LIN {X 0,Y 474.319,Z 459.173,A -85,B 0,C 180,E1 -7298.735,E2 -7298.735} C_VEL
LIN {X 0,Y 474.674,Z 450.889,A -85,B 0,C 180,E1 -7300.018,E2 -7300.018} C_VEL
LIN {X 0,Y 475.05,Z 442.392,A -85,B 0,C 180,E1 -7301.088,E2 -7301.088} C_VEL
LIN {X 0,Y 475.606,Z 432.048,A -85,B 0,C 180,E1 -7302.141,E2 -7302.141} C_VEL
LIN {X 0,Y 475.98,Z 420.23,A -85,B 0,C 180,E1 -7303.109,E2 -7303.109} C_VEL
LIN {X 0,Y 476.476,Z 408.181,A -85,B 0,C 180,E1 -7303.867,E2 -7303.867} C_VEL
LIN {X 0,Y 476.914,Z 395.801,A -85,B 0,C 180,E1 -7304.453,E2 -7304.453} C_VEL
LIN {X 0,Y 477.291,Z 383.062,A -85,B 0,C 180,E1 -7304.877,E2 -7304.877} C_VEL
LIN {X 0,Y 477.535,Z 367.874,A -85,B 0,C 180,E1 -7305.17,E2 -7305.17} C_VEL
LIN {X 0,Y 478.066,Z 286.385,A -85,B 0,C 180,E1 -7306.413,E2 -7306.413} C_VEL
LIN {X 0,Y 475.418,Z 270.175,A -85,B 0,C 180,E1 -7306.789,E2 -7306.789} C_VEL
LIN {X 0,Y 475.587,Z 262.703,A -85,B 0,C 180,E1 -7308.078,E2 -7308.078} C_VEL
LIN {X 0,Y 476.357,Z 243.825,A -85,B 0,C 180,E1 -7311.518,E2 -7311.518} C_VEL
LIN {X 0,Y 476.393,Z 237.035,A -85,B 0,C 180,E1 -7312.783,E2 -7312.783} C_VEL
LIN {X 0,Y 474.661,Z 227.951,A -85,B 0,C 180,E1 -7314.637,E2 -7314.637} C_VEL
LIN {X 0,Y 474.679,Z 227.858,A -85,B 0,C 180,E1 -7317.331,E2 -7317.331} C_VEL
LIN {X 0,Y 474.608,Z 227.867,A -85,B 0,C 180,E1 -7320.229,E2 -7320.229} C_VEL
LIN {X 0,Y 474.638,Z 227.86,A -85,B 0,C 180,E1 -7323.219,E2 -7323.219} C_VEL
LIN {X 0,Y 474.587,Z 227.865,A -85,B 0,C 180,E1 -7326.322,E2 -7326.322} C_VEL
LIN {X 0,Y 474.624,Z 227.861,A -85,B 0,C 180,E1 -7329.547,E2 -7329.547} C_VEL
LIN {X 0,Y 474.6,Z 227.87,A -85,B 0,C 180,E1 -7332.231,E2 -7332.231} C_VEL
LIN {X 0,Y 474.618,Z 227.86,A -85,B 0,C 180,E1 -7335.296,E2 -7335.296} C_VEL
LIN {X 0,Y 474.61,Z 227.867,A -85,B 0,C 180,E1 -7338.211,E2 -7338.211} C_VEL
LIN {X 0,Y 474.609,Z 227.858,A -85,B 0,C 180,E1 -7341.54,E2 -7341.54} C_VEL
LIN {X 0,Y 474.619,Z 227.864,A -85,B 0,C 180,E1 -7344.723,E2 -7344.723} C_VEL
LIN {X 0,Y 474.627,Z 227.858,A -85,B 0,C 180,E1 -7347.785,E2 -7347.785} C_VEL
LIN {X 0,Y 474.597,Z 227.868,A -85,B 0,C 180,E1 -7350.888,E2 -7350.888} C_VEL
LIN {X 0,Y 474.588,Z 227.863,A -85,B 0,C 180,E1 -7353.622,E2 -7353.622} C_VEL
LIN {X 0,Y 474.632,Z 227.862,A -85,B 0,C 180,E1 -7356.64,E2 -7356.64} C_VEL
LIN {X 0,Y 474.646,Z 227.856,A -85,B 0,C 180,E1 -7360.087,E2 -7360.087} C_VEL
LIN {X 0,Y 474.628,Z 227.859,A -85,B 0,C 180,E1 -7362.771,E2 -7362.771} C_VEL
LIN {X 0,Y 474.627,Z 227.86,A -85,B 0,C 180,E1 -7365.418,E2 -7365.418} C_VEL
LIN {X 0,Y 474.698,Z 227.849,A -85,B 0,C 180,E1 -7368.035,E2 -7368.035} C_VEL
LIN {X 0,Y 474.66,Z 227.857,A -85,B 0,C 180,E1 -7371.483,E2 -7371.483} C_VEL
LIN {X 0,Y 474.748,Z 227.845,A -85,B 0,C 180,E1 -7374.049,E2 -7374.049} C_VEL
LIN {X 0,Y 474.859,Z 227.833,A -85,B 0,C 180,E1 -7377.452,E2 -7377.452} C_VEL
LIN {X 0,Y 474.865,Z 227.829,A -85,B 0,C 180,E1 -7379.997,E2 -7379.997} C_VEL
LIN {X 0,Y 474.833,Z 227.833,A -85,B 0,C 180,E1 -7382.542,E2 -7382.542} C_VEL
LIN {X 0,Y 474.714,Z 227.852,A -85,B 0,C 180,E1 -7385.945,E2 -7385.945} C_VEL
LIN {X 0,Y 474.65,Z 227.856,A -85,B 0,C 180,E1 -7388.512,E2 -7388.512} C_VEL
LIN {X 0,Y 474.678,Z 227.86,A -85,B 0,C 180,E1 -7391.96,E2 -7391.96} C_VEL
LIN {X 0,Y 474.681,Z 227.855,A -85,B 0,C 180,E1 -7395.453,E2 -7395.453} C_VEL
LIN {X 0,Y 474.642,Z 227.858,A -85,B 0,C 180,E1 -7399.007,E2 -7399.007} C_VEL
LIN {X 0,Y 474.568,Z 227.869,A -85,B 0,C 180,E1 -7401.726,E2 -7401.726} C_VEL
LIN {X 0,Y 474.615,Z 227.865,A -85,B 0,C 180,E1 -7404.491,E2 -7404.491} C_VEL
LIN {X 0,Y 474.614,Z 227.861,A -85,B 0,C 180,E1 -7407.321,E2 -7407.321} C_VEL
LIN {X 0,Y 474.578,Z 227.87,A -85,B 0,C 180,E1 -7410.228,E2 -7410.228} C_VEL
LIN {X 0,Y 474.617,Z 227.862,A -85,B 0,C 180,E1 -7413.217,E2 -7413.217} C_VEL
LIN {X 0,Y 474.566,Z 227.872,A -85,B 0,C 180,E1 -7416.321,E2 -7416.321} C_VEL
LIN {X 0,Y 474.622,Z 227.862,A -85,B 0,C 180,E1 -7419.648,E2 -7419.648} C_VEL
LIN {X 0,Y 474.623,Z 227.867,A -85,B 0,C 180,E1 -7422.928,E2 -7422.928} C_VEL
LIN {X 0,Y 474.644,Z 227.955,A -85,B 0,C 180,E1 -7424.526,E2 -7424.526} C_VEL
LIN {X 0,Y 475.947,Z 235.272,A -85,B 0,C 180,E1 -7426.052,E2 -7426.052} C_VEL
LIN {X 0,Y 475.635,Z 249.047,A -85,B 0,C 180,E1 -7428.661,E2 -7428.661} C_VEL
LIN {X 0,Y 475.424,Z 257.75,A -85,B 0,C 180,E1 -7430.256,E2 -7430.256} C_VEL
LIN {X 0,Y 478.108,Z 273.113,A -85,B 0,C 180,E1 -7430.623,E2 -7430.623} C_VEL
LIN {X 0,Y 477.39,Z 365.589,A -85,B 0,C 180,E1 -7432.055,E2 -7432.055} C_VEL
LIN {X 0,Y 477.099,Z 378.912,A -85,B 0,C 180,E1 -7432.436,E2 -7432.436} C_VEL
LIN {X 0,Y 476.816,Z 391.076,A -85,B 0,C 180,E1 -7432.954,E2 -7432.954} C_VEL
LIN {X 0,Y 476.403,Z 402.075,A -85,B 0,C 180,E1 -7433.576,E2 -7433.576} C_VEL
LIN {X 0,Y 476.121,Z 407.981,A -85,B 0,C 180,E1 -7433.98,E2 -7433.98} C_VEL
LIN {X 0,Y 475.228,Z 413.061,A -85,B 0,C 180,E1 -7434.352,E2 -7434.352} C_VEL
LIN {X 0,Y 472.047,Z 420.996,A -85,B 0,C 180,E1 -7434.971,E2 -7434.971} C_VEL
LIN {X 0,Y 468.888,Z 428.372,A -85,B 0,C 180,E1 -7435.666,E2 -7435.666} C_VEL
LIN {X 0,Y 468.021,Z 432.578,A -85,B 0,C 180,E1 -7436.148,E2 -7436.148} C_VEL
LIN {X 0,Y 467.606,Z 441.038,A -85,B 0,C 180,E1 -7437.308,E2 -7437.308} C_VEL
LIN {X 0,Y 467.237,Z 449.029,A -85,B 0,C 180,E1 -7438.674,E2 -7438.674} C_VEL
LIN {X 0,Y 467.002,Z 455.116,A -85,B 0,C 180,E1 -7439.976,E2 -7439.976} C_VEL
LIN {X 0,Y 466.824,Z 459.697,A -85,B 0,C 180,E1 -7441.201,E2 -7441.201} C_VEL
LIN {X 0,Y 466.694,Z 463.897,A -85,B 0,C 180,E1 -7442.674,E2 -7442.674} C_VEL
LIN {X 0,Y 466.564,Z 466.729,A -85,B 0,C 180,E1 -7444.099,E2 -7444.099} C_VEL
LIN {X 0,Y 466.508,Z 467.992,A -85,B 0,C 180,E1 -7445.051,E2 -7445.051} C_VEL
LIN {X 0,Y 466.486,Z 469.005,A -85,B 0,C 180,E1 -7446.771,E2 -7446.771} C_VEL
LIN {X 0,Y 466.467,Z 468.848,A -85,B 0,C 180,E1 -7447.874,E2 -7447.874} C_VEL
LIN {X 0,Y 466.511,Z 467.954,A -85,B 0,C 180,E1 -7449.059,E2 -7449.059} C_VEL
LIN {X 0,Y 466.617,Z 465.531,A -85,B 0,C 180,E1 -7450.65,E2 -7450.65} C_VEL
LIN {X 0,Y 466.715,Z 462.294,A -85,B 0,C 180,E1 -7452.02,E2 -7452.02} C_VEL
LIN {X 0,Y 466.863,Z 457.92,A -85,B 0,C 180,E1 -7453.381,E2 -7453.381} C_VEL
LIN {X 0,Y 467.122,Z 452.119,A -85,B 0,C 180,E1 -7454.772,E2 -7454.772} C_VEL
LIN {X 0,Y 467.411,Z 445.255,A -85,B 0,C 180,E1 -7456.08,E2 -7456.08} C_VEL
LIN {X 0,Y 467.793,Z 437.03,A -85,B 0,C 180,E1 -7457.34,E2 -7457.34} C_VEL
LIN {X 0,Y 468.253,Z 427.374,A -85,B 0,C 180,E1 -7458.53,E2 -7458.53} C_VEL
LIN {X 0,Y 468.76,Z 417.39,A -85,B 0,C 180,E1 -7459.527,E2 -7459.527} C_VEL
LIN {X 0,Y 469.247,Z 406.384,A -85,B 0,C 180,E1 -7460.409,E2 -7460.409} C_VEL
LIN {X 0,Y 469.753,Z 394.705,A -85,B 0,C 180,E1 -7461.14,E2 -7461.14} C_VEL
LIN {X 0,Y 470.088,Z 382.336,A -85,B 0,C 180,E1 -7461.727,E2 -7461.727} C_VEL
LIN {X 0,Y 470.482,Z 369.805,A -85,B 0,C 180,E1 -7462.14,E2 -7462.14} C_VEL
LIN {X 0,Y 470.668,Z 355.83,A -85,B 0,C 180,E1 -7462.412,E2 -7462.412} C_VEL
LIN {X 0,Y 471.164,Z 272.816,A -85,B 0,C 180,E1 -7463.698,E2 -7463.698} C_VEL
LIN {X 0,Y 468.501,Z 258.149,A -85,B 0,C 180,E1 -7464.054,E2 -7464.054} C_VEL
LIN {X 0,Y 468.635,Z 252.883,A -85,B 0,C 180,E1 -7465.054,E2 -7465.054} C_VEL
LIN {X 0,Y 469.214,Z 238.012,A -85,B 0,C 180,E1 -7468.069,E2 -7468.069} C_VEL
LIN {X 0,Y 467.876,Z 229.061,A -85,B 0,C 180,E1 -7470.001,E2 -7470.001} C_VEL
LIN {X 0,Y 467.826,Z 228.707,A -85,B 0,C 180,E1 -7470.216,E2 -7470.216} C_VEL
LIN {X 0,Y 467.822,Z 228.711,A -85,B 0,C 180,E1 -7472.584,E2 -7472.584} C_VEL
LIN {X 0,Y 467.706,Z 228.723,A -85,B 0,C 180,E1 -7476.039,E2 -7476.039} C_VEL
LIN {X 0,Y 467.644,Z 228.73,A -85,B 0,C 180,E1 -7478.644,E2 -7478.644} C_VEL
LIN {X 0,Y 467.646,Z 228.726,A -85,B 0,C 180,E1 -7482.146,E2 -7482.146} C_VEL
LIN {X 0,Y 467.613,Z 228.737,A -85,B 0,C 180,E1 -7485.887,E2 -7485.887} C_VEL
LIN {X 0,Y 467.588,Z 228.737,A -85,B 0,C 180,E1 -7489.31,E2 -7489.31} C_VEL
LIN {X 0,Y 467.5,Z 228.754,A -85,B 0,C 180,E1 -7492.076,E2 -7492.076} C_VEL
LIN {X 0,Y 467.55,Z 228.739,A -85,B 0,C 180,E1 -7494.891,E2 -7494.891} C_VEL
LIN {X 0,Y 467.548,Z 228.744,A -85,B 0,C 180,E1 -7497.774,E2 -7497.774} C_VEL
LIN {X 0,Y 467.537,Z 228.742,A -85,B 0,C 180,E1 -7501.047,E2 -7501.047} C_VEL
LIN {X 0,Y 467.546,Z 228.744,A -85,B 0,C 180,E1 -7504.243,E2 -7504.243} C_VEL
LIN {X 0,Y 467.493,Z 228.747,A -85,B 0,C 180,E1 -7507.185,E2 -7507.185} C_VEL
LIN {X 0,Y 467.529,Z 228.747,A -85,B 0,C 180,E1 -7510.27,E2 -7510.27} C_VEL
LIN {X 0,Y 467.521,Z 228.738,A -85,B 0,C 180,E1 -7513.749,E2 -7513.749} C_VEL
LIN {X 0,Y 467.521,Z 228.745,A -85,B 0,C 180,E1 -7516.258,E2 -7516.258} C_VEL
LIN {X 0,Y 467.536,Z 228.735,A -85,B 0,C 180,E1 -7519.737,E2 -7519.737} C_VEL
LIN {X 0,Y 467.528,Z 228.739,A -85,B 0,C 180,E1 -7522.818,E2 -7522.818} C_VEL
LIN {X 0,Y 467.56,Z 228.739,A -85,B 0,C 180,E1 -7525.764,E2 -7525.764} C_VEL
LIN {X 0,Y 467.528,Z 228.746,A -85,B 0,C 180,E1 -7528.964,E2 -7528.964} C_VEL
LIN {X 0,Y 467.53,Z 228.731,A -85,B 0,C 180,E1 -7532.23,E2 -7532.23} C_VEL
LIN {X 0,Y 467.542,Z 228.742,A -85,B 0,C 180,E1 -7535.113,E2 -7535.113} C_VEL
LIN {X 0,Y 467.522,Z 228.744,A -85,B 0,C 180,E1 -7537.93,E2 -7537.93} C_VEL
LIN {X 0,Y 467.612,Z 228.724,A -85,B 0,C 180,E1 -7540.696,E2 -7540.696} C_VEL
LIN {X 0,Y 467.632,Z 228.724,A -85,B 0,C 180,E1 -7544.308,E2 -7544.308} C_VEL
LIN {X 0,Y 467.644,Z 228.736,A -85,B 0,C 180,E1 -7547.858,E2 -7547.858} C_VEL
LIN {X 0,Y 467.653,Z 228.725,A -85,B 0,C 180,E1 -7551.36,E2 -7551.36} C_VEL
LIN {X 0,Y 467.701,Z 228.711,A -85,B 0,C 180,E1 -7553.965,E2 -7553.965} C_VEL
LIN {X 0,Y 467.813,Z 228.703,A -85,B 0,C 180,E1 -7557.42,E2 -7557.42} C_VEL
LIN {X 0,Y 467.849,Z 228.708,A -85,B 0,C 180,E1 -7560.003,E2 -7560.003} C_VEL
LIN {X 0,Y 467.814,Z 228.704,A -85,B 0,C 180,E1 -7562.586,E2 -7562.586} C_VEL
LIN {X 0,Y 467.718,Z 228.708,A -85,B 0,C 180,E1 -7566.04,E2 -7566.04} C_VEL
LIN {X 0,Y 467.663,Z 228.732,A -85,B 0,C 180,E1 -7568.646,E2 -7568.646} C_VEL
LIN {X 0,Y 467.662,Z 228.728,A -85,B 0,C 180,E1 -7572.148,E2 -7572.148} C_VEL
LIN {X 0,Y 467.656,Z 228.716,A -85,B 0,C 180,E1 -7575.887,E2 -7575.887} C_VEL
LIN {X 0,Y 467.629,Z 228.733,A -85,B 0,C 180,E1 -7579.31,E2 -7579.31} C_VEL
LIN {X 0,Y 467.539,Z 228.739,A -85,B 0,C 180,E1 -7582.076,E2 -7582.076} C_VEL
LIN {X 0,Y 467.577,Z 228.733,A -85,B 0,C 180,E1 -7584.891,E2 -7584.891} C_VEL
LIN {X 0,Y 467.571,Z 228.738,A -85,B 0,C 180,E1 -7587.774,E2 -7587.774} C_VEL
LIN {X 0,Y 467.574,Z 228.738,A -85,B 0,C 180,E1 -7591.045,E2 -7591.045} C_VEL
LIN {X 0,Y 467.586,Z 228.736,A -85,B 0,C 180,E1 -7594.241,E2 -7594.241} C_VEL
LIN {X 0,Y 467.552,Z 228.743,A -85,B 0,C 180,E1 -7597.186,E2 -7597.186} C_VEL
LIN {X 0,Y 467.569,Z 228.738,A -85,B 0,C 180,E1 -7600.268,E2 -7600.268} C_VEL
LIN {X 0,Y 467.553,Z 228.735,A -85,B 0,C 180,E1 -7602.566,E2 -7602.566} C_VEL
LIN {X 0,Y 467.575,Z 228.739,A -85,B 0,C 180,E1 -7605.053,E2 -7605.053} C_VEL
LIN {X 0,Y 467.574,Z 228.737,A -85,B 0,C 180,E1 -7608.726,E2 -7608.726} C_VEL
LIN {X 0,Y 467.571,Z 228.744,A -85,B 0,C 180,E1 -7611.956,E2 -7611.956} C_VEL
LIN {X 0,Y 467.572,Z 228.739,A -85,B 0,C 180,E1 -7615.168,E2 -7615.168} C_VEL
LIN {X 0,Y 467.592,Z 228.741,A -85,B 0,C 180,E1 -7618.26,E2 -7618.26} C_VEL
LIN {X 0,Y 467.582,Z 228.738,A -85,B 0,C 180,E1 -7621.25,E2 -7621.25} C_VEL
LIN {X 0,Y 467.597,Z 228.743,A -85,B 0,C 180,E1 -7624.159,E2 -7624.159} C_VEL
LIN {X 0,Y 467.654,Z 228.952,A -85,B 0,C 180,E1 -7625.115,E2 -7625.115} C_VEL
LIN {X 0,Y 469.616,Z 239.761,A -85,B 0,C 180,E1 -7627.333,E2 -7627.333} C_VEL
LIN {X 0,Y 469.166,Z 250.64,A -85,B 0,C 180,E1 -7629.388,E2 -7629.388} C_VEL
LIN {X 0,Y 468.53,Z 266.336,A -85,B 0,C 180,E1 -7632.316,E2 -7632.316} C_VEL
LIN {X 0,Y 468.406,Z 270.181,A -85,B 0,C 180,E1 -7632.979,E2 -7632.979} C_VEL
LIN {X 0,Y 471.24,Z 287.662,A -85,B 0,C 180,E1 -7633.384,E2 -7633.384} C_VEL
LIN {X 0,Y 470.546,Z 377.761,A -85,B 0,C 180,E1 -7634.792,E2 -7634.792} C_VEL
LIN {X 0,Y 470.203,Z 391.031,A -85,B 0,C 180,E1 -7635.169,E2 -7635.169} C_VEL
LIN {X 0,Y 469.781,Z 403.762,A -85,B 0,C 180,E1 -7635.709,E2 -7635.709} C_VEL
LIN {X 0,Y 469.301,Z 415.395,A -85,B 0,C 180,E1 -7636.379,E2 -7636.379} C_VEL
LIN {X 0,Y 468.806,Z 426.182,A -85,B 0,C 180,E1 -7637.176,E2 -7637.176} C_VEL
LIN {X 0,Y 468.289,Z 437.241,A -85,B 0,C 180,E1 -7638.2,E2 -7638.2} C_VEL
LIN {X 0,Y 467.866,Z 445.818,A -85,B 0,C 180,E1 -7639.177,E2 -7639.177} C_VEL
LIN {X 0,Y 467.483,Z 453.726,A -85,B 0,C 180,E1 -7640.262,E2 -7640.262} C_VEL
LIN {X 0,Y 467.154,Z 461.449,A -85,B 0,C 180,E1 -7641.565,E2 -7641.565} C_VEL
LIN {X 0,Y 466.86,Z 468.553,A -85,B 0,C 180,E1 -7643.082,E2 -7643.082} C_VEL
LIN {X 0,Y 466.792,Z 473.281,A -85,B 0,C 180,E1 -7644.383,E2 -7644.383} C_VEL
LIN {X 0,Y 466.649,Z 476.891,A -85,B 0,C 180,E1 -7645.681,E2 -7645.681} C_VEL
LIN {X 0,Y 466.663,Z 478.755,A -85,B 0,C 180,E1 -7646.546,E2 -7646.546} C_VEL
LIN {X 0,Y 466.646,Z 480.152,A -85,B 0,C 180,E1 -7647.41,E2 -7647.41} C_VEL
LIN {X 0,Y 466.591,Z 481.755,A -85,B 0,C 180,E1 -7649.136,E2 -7649.136} C_VEL
LIN {X 0,Y 466.601,Z 481.973,A -85,B 0,C 180,E1 -7649.999,E2 -7649.999} C_VEL
LIN {X 0,Y 466.606,Z 481.151,A -85,B 0,C 180,E1 -7651.726,E2 -7651.726} C_VEL
LIN {X 0,Y 466.646,Z 480.157,A -85,B 0,C 180,E1 -7652.589,E2 -7652.589} C_VEL
LIN {X 0,Y 466.663,Z 478.763,A -85,B 0,C 180,E1 -7653.453,E2 -7653.453} C_VEL
LIN {X 0,Y 466.693,Z 475.829,A -85,B 0,C 180,E1 -7654.75,E2 -7654.75} C_VEL
LIN {X 0,Y 466.78,Z 471.859,A -85,B 0,C 180,E1 -7656.049,E2 -7656.049} C_VEL
LIN {X 0,Y 466.981,Z 465.754,A -85,B 0,C 180,E1 -7657.566,E2 -7657.566} C_VEL
LIN {X 0,Y 467.282,Z 459.082,A -85,B 0,C 180,E1 -7658.867,E2 -7658.867} C_VEL
LIN {X 0,Y 467.63,Z 450.802,A -85,B 0,C 180,E1 -7660.17,E2 -7660.17} C_VEL
LIN {X 0,Y 468.068,Z 442.312,A -85,B 0,C 180,E1 -7661.255,E2 -7661.255} C_VEL
LIN {X 0,Y 468.648,Z 432.148,A -85,B 0,C 180,E1 -7662.308,E2 -7662.308} C_VEL
LIN {X 0,Y 468.971,Z 421.726,A -85,B 0,C 180,E1 -7663.188,E2 -7663.188} C_VEL
LIN {X 0,Y 469.522,Z 410.055,A -85,B 0,C 180,E1 -7663.966,E2 -7663.966} C_VEL
LIN {X 0,Y 469.958,Z 398.351,A -85,B 0,C 180,E1 -7664.561,E2 -7664.561} C_VEL
LIN {X 0,Y 470.425,Z 384.874,A -85,B 0,C 180,E1 -7665.044,E2 -7665.044} C_VEL
LIN {X 0,Y 470.647,Z 371.473,A -85,B 0,C 180,E1 -7665.342,E2 -7665.342} C_VEL
LIN {X 0,Y 471.274,Z 287.31,A -85,B 0,C 180,E1 -7666.643,E2 -7666.643} C_VEL
LIN {X 0,Y 468.443,Z 270.181,A -85,B 0,C 180,E1 -7667.044,E2 -7667.044} C_VEL
LIN {X 0,Y 468.441,Z 267.494,A -85,B 0,C 180,E1 -7667.46,E2 -7667.46} C_VEL
LIN {X 0,Y 469.125,Z 250.395,A -85,B 0,C 180,E1 -7670.612,E2 -7670.612} C_VEL
LIN {X 0,Y 469.575,Z 239.398,A -85,B 0,C 180,E1 -7672.667,E2 -7672.667} C_VEL
LIN {X 0,Y 467.644,Z 228.871,A -85,B 0,C 180,E1 -7674.825,E2 -7674.825} C_VEL
LIN {X 0,Y 467.621,Z 228.739,A -85,B 0,C 180,E1 -7677.768,E2 -7677.768} C_VEL
LIN {X 0,Y 467.571,Z 228.741,A -85,B 0,C 180,E1 -7681.043,E2 -7681.043} C_VEL
LIN {X 0,Y 467.592,Z 228.741,A -85,B 0,C 180,E1 -7684.24,E2 -7684.24} C_VEL
LIN {X 0,Y 467.545,Z 228.739,A -85,B 0,C 180,E1 -7687.184,E2 -7687.184} C_VEL
LIN {X 0,Y 467.562,Z 228.74,A -85,B 0,C 180,E1 -7690.265,E2 -7690.265} C_VEL
LIN {X 0,Y 467.563,Z 228.742,A -85,B 0,C 180,E1 -7692.562,E2 -7692.562} C_VEL
LIN {X 0,Y 467.567,Z 228.739,A -85,B 0,C 180,E1 -7695.051,E2 -7695.051} C_VEL
LIN {X 0,Y 467.568,Z 228.744,A -85,B 0,C 180,E1 -7698.594,E2 -7698.594} C_VEL
LIN {X 0,Y 467.562,Z 228.738,A -85,B 0,C 180,E1 -7701.953,E2 -7701.953} C_VEL
LIN {X 0,Y 467.556,Z 228.74,A -85,B 0,C 180,E1 -7705.164,E2 -7705.164} C_VEL
LIN {X 0,Y 467.577,Z 228.74,A -85,B 0,C 180,E1 -7708.257,E2 -7708.257} C_VEL
LIN {X 0,Y 467.543,Z 228.742,A -85,B 0,C 180,E1 -7711.246,E2 -7711.246} C_VEL
LIN {X 0,Y 467.576,Z 228.739,A -85,B 0,C 180,E1 -7714.399,E2 -7714.399} C_VEL
LIN {X 0,Y 467.57,Z 228.74,A -85,B 0,C 180,E1 -7716.993,E2 -7716.993} C_VEL
LIN {X 0,Y 467.617,Z 228.732,A -85,B 0,C 180,E1 -7719.775,E2 -7719.775} C_VEL
LIN {X 0,Y 467.589,Z 228.733,A -85,B 0,C 180,E1 -7722.504,E2 -7722.504} C_VEL
LIN {X 0,Y 467.589,Z 228.74,A -85,B 0,C 180,E1 -7725.193,E2 -7725.193} C_VEL
LIN {X 0,Y 467.65,Z 228.728,A -85,B 0,C 180,E1 -7727.852,E2 -7727.852} C_VEL
LIN {X 0,Y 467.629,Z 228.732,A -85,B 0,C 180,E1 -7731.354,E2 -7731.354} C_VEL
LIN {X 0,Y 467.713,Z 228.722,A -85,B 0,C 180,E1 -7733.959,E2 -7733.959} C_VEL
LIN {X 0,Y 467.8,Z 228.712,A -85,B 0,C 180,E1 -7737.414,E2 -7737.414} C_VEL
LIN {X 0,Y 467.814,Z 228.707,A -85,B 0,C 180,E1 -7739.997,E2 -7739.997} C_VEL
LIN {X 0,Y 467.777,Z 228.712,A -85,B 0,C 180,E1 -7742.58,E2 -7742.58} C_VEL
LIN {X 0,Y 467.679,Z 228.728,A -85,B 0,C 180,E1 -7746.035,E2 -7746.035} C_VEL
LIN {X 0,Y 467.619,Z 228.731,A -85,B 0,C 180,E1 -7748.641,E2 -7748.641} C_VEL
LIN {X 0,Y 467.632,Z 228.735,A -85,B 0,C 180,E1 -7752.143,E2 -7752.143} C_VEL
LIN {X 0,Y 467.621,Z 228.737,A -85,B 0,C 180,E1 -7755.692,E2 -7755.692} C_VEL
LIN {X 0,Y 467.601,Z 228.735,A -85,B 0,C 180,E1 -7759.305,E2 -7759.305} C_VEL
LIN {X 0,Y 467.515,Z 228.753,A -85,B 0,C 180,E1 -7762.071,E2 -7762.071} C_VEL
LIN {X 0,Y 467.562,Z 228.739,A -85,B 0,C 180,E1 -7764.886,E2 -7764.886} C_VEL
LIN {X 0,Y 467.558,Z 228.742,A -85,B 0,C 180,E1 -7767.769,E2 -7767.769} C_VEL
LIN {X 0,Y 467.543,Z 228.743,A -85,B 0,C 180,E1 -7771.042,E2 -7771.042} C_VEL
LIN {X 0,Y 467.564,Z 228.745,A -85,B 0,C 180,E1 -7774.24,E2 -7774.24} C_VEL
LIN {X 0,Y 467.523,Z 228.746,A -85,B 0,C 180,E1 -7777.184,E2 -7777.184} C_VEL
LIN {X 0,Y 467.568,Z 228.744,A -85,B 0,C 180,E1 -7780.26,E2 -7780.26} C_VEL
LIN {X 0,Y 467.59,Z 228.742,A -85,B 0,C 180,E1 -7782.569,E2 -7782.569} C_VEL
LIN {X 0,Y 467.591,Z 228.848,A -85,B 0,C 180,E1 -7784.341,E2 -7784.341} C_VEL
LIN {X 0,Y 469.033,Z 236.661,A -85,B 0,C 180,E1 -7785.985,E2 -7785.985} C_VEL
LIN {X 0,Y 468.672,Z 250.101,A -85,B 0,C 180,E1 -7788.564,E2 -7788.564} C_VEL
LIN {X 0,Y 468.47,Z 257.854,A -85,B 0,C 180,E1 -7789.993,E2 -7789.993} C_VEL
LIN {X 0,Y 470.658,Z 269.971,A -85,B 0,C 180,E1 -7790.3,E2 -7790.3} C_VEL
LIN {X 0,Y 471.343,Z 275.192,A -85,B 0,C 180,E1 -7790.409,E2 -7790.409} C_VEL
LIN {X 0,Y 470.548,Z 365.863,A -85,B 0,C 180,E1 -7791.833,E2 -7791.833} C_VEL
LIN {X 0,Y 470.245,Z 379.37,A -85,B 0,C 180,E1 -7792.23,E2 -7792.23} C_VEL
LIN {X 0,Y 469.899,Z 392.099,A -85,B 0,C 180,E1 -7792.787,E2 -7792.787} C_VEL
LIN {X 0,Y 469.448,Z 403.23,A -85,B 0,C 180,E1 -7793.443,E2 -7793.443} C_VEL
LIN {X 0,Y 468.858,Z 415.313,A -85,B 0,C 180,E1 -7794.359,E2 -7794.359} C_VEL
LIN {X 0,Y 468.382,Z 425.748,A -85,B 0,C 180,E1 -7795.358,E2 -7795.358} C_VEL
LIN {X 0,Y 468.021,Z 432.578,A -85,B 0,C 180,E1 -7796.148,E2 -7796.148} C_VEL
LIN {X 0,Y 467.149,Z 436.69,A -85,B 0,C 180,E1 -7796.659,E2 -7796.659} C_VEL
LIN {X 0,Y 463.971,Z 443.007,A -85,B 0,C 180,E1 -7797.519,E2 -7797.519} C_VEL
LIN {X 0,Y 460.852,Z 448.667,A -85,B 0,C 180,E1 -7798.452,E2 -7798.452} C_VEL
LIN {X 0,Y 460.083,Z 451.747,A -85,B 0,C 180,E1 -7799.073,E2 -7799.073} C_VEL
LIN {X 0,Y 459.818,Z 458.017,A -85,B 0,C 180,E1 -7800.589,E2 -7800.589} C_VEL
LIN {X 0,Y 459.649,Z 462.837,A -85,B 0,C 180,E1 -7802.13,E2 -7802.13} C_VEL
LIN {X 0,Y 459.496,Z 466.202,A -85,B 0,C 180,E1 -7803.67,E2 -7803.67} C_VEL
LIN {X 0,Y 459.448,Z 467.646,A -85,B 0,C 180,E1 -7804.641,E2 -7804.641} C_VEL
LIN {X 0,Y 459.388,Z 468.621,A -85,B 0,C 180,E1 -7805.604,E2 -7805.604} C_VEL
LIN {X 0,Y 459.385,Z 469.077,A -85,B 0,C 180,E1 -7806.612,E2 -7806.612} C_VEL
LIN {X 0,Y 459.369,Z 469.065,A -85,B 0,C 180,E1 -7807.514,E2 -7807.514} C_VEL
LIN {X 0,Y 459.42,Z 468.206,A -85,B 0,C 180,E1 -7808.918,E2 -7808.918} C_VEL
LIN {X 0,Y 459.508,Z 466.289,A -85,B 0,C 180,E1 -7810.338,E2 -7810.338} C_VEL
LIN {X 0,Y 459.601,Z 464.045,A -85,B 0,C 180,E1 -7811.44,E2 -7811.44} C_VEL
LIN {X 0,Y 459.738,Z 459.279,A -85,B 0,C 180,E1 -7813.116,E2 -7813.116} C_VEL
LIN {X 0,Y 460.015,Z 453.486,A -85,B 0,C 180,E1 -7814.609,E2 -7814.609} C_VEL
LIN {X 0,Y 460.337,Z 446.061,A -85,B 0,C 180,E1 -7816.087,E2 -7816.087} C_VEL
LIN {X 0,Y 460.768,Z 437.468,A -85,B 0,C 180,E1 -7817.446,E2 -7817.446} C_VEL
LIN {X 0,Y 461.216,Z 428.58,A -85,B 0,C 180,E1 -7818.575,E2 -7818.575} C_VEL
LIN {X 0,Y 461.806,Z 417.615,A -85,B 0,C 180,E1 -7819.7,E2 -7819.7} C_VEL
LIN {X 0,Y 462.317,Z 407.003,A -85,B 0,C 180,E1 -7820.57,E2 -7820.57} C_VEL
LIN {X 0,Y 462.842,Z 395.275,A -85,B 0,C 180,E1 -7821.322,E2 -7821.322} C_VEL
LIN {X 0,Y 463.211,Z 382.698,A -85,B 0,C 180,E1 -7821.933,E2 -7821.933} C_VEL
LIN {X 0,Y 463.64,Z 370.292,A -85,B 0,C 180,E1 -7822.352,E2 -7822.352} C_VEL
LIN {X 0,Y 463.817,Z 356.646,A -85,B 0,C 180,E1 -7822.628,E2 -7822.628} C_VEL
LIN {X 0,Y 464.339,Z 273.699,A -85,B 0,C 180,E1 -7823.933,E2 -7823.933} C_VEL
LIN {X 0,Y 461.578,Z 258.553,A -85,B 0,C 180,E1 -7824.294,E2 -7824.294} C_VEL
LIN {X 0,Y 461.552,Z 257.413,A -85,B 0,C 180,E1 -7824.43,E2 -7824.43} C_VEL
LIN {X 0,Y 462.272,Z 240.826,A -85,B 0,C 180,E1 -7827.823,E2 -7827.823} C_VEL
LIN {X 0,Y 461.62,Z 234.738,A -85,B 0,C 180,E1 -7829.128,E2 -7829.128} C_VEL
LIN {X 0,Y 460.796,Z 229.649,A -85,B 0,C 180,E1 -7830.301,E2 -7830.301} C_VEL
LIN {X 0,Y 460.788,Z 229.588,A -85,B 0,C 180,E1 -7832.623,E2 -7832.623} C_VEL
LIN {X 0,Y 460.671,Z 229.599,A -85,B 0,C 180,E1 -7836.131,E2 -7836.131} C_VEL
LIN {X 0,Y 460.591,Z 229.609,A -85,B 0,C 180,E1 -7838.778,E2 -7838.778} C_VEL
LIN {X 0,Y 460.598,Z 229.602,A -85,B 0,C 180,E1 -7842.458,E2 -7842.458} C_VEL
LIN {X 0,Y 460.565,Z 229.614,A -85,B 0,C 180,E1 -7845.999,E2 -7845.999} C_VEL
LIN {X 0,Y 460.536,Z 229.614,A -85,B 0,C 180,E1 -7848.903,E2 -7848.903} C_VEL
LIN {X 0,Y 460.482,Z 229.622,A -85,B 0,C 180,E1 -7851.488,E2 -7851.488} C_VEL
LIN {X 0,Y 460.496,Z 229.622,A -85,B 0,C 180,E1 -7854.335,E2 -7854.335} C_VEL
LIN {X 0,Y 460.502,Z 229.618,A -85,B 0,C 180,E1 -7857.249,E2 -7857.249} C_VEL
LIN {X 0,Y 460.476,Z 229.623,A -85,B 0,C 180,E1 -7860.243,E2 -7860.243} C_VEL
LIN {X 0,Y 460.487,Z 229.619,A -85,B 0,C 180,E1 -7863.329,E2 -7863.329} C_VEL
LIN {X 0,Y 460.436,Z 229.629,A -85,B 0,C 180,E1 -7866.534,E2 -7866.534} C_VEL
LIN {X 0,Y 460.483,Z 229.621,A -85,B 0,C 180,E1 -7869.868,E2 -7869.868} C_VEL
LIN {X 0,Y 460.442,Z 229.623,A -85,B 0,C 180,E1 -7872.897,E2 -7872.897} C_VEL
LIN {X 0,Y 460.48,Z 229.62,A -85,B 0,C 180,E1 -7875.835,E2 -7875.835} C_VEL
LIN {X 0,Y 460.493,Z 229.619,A -85,B 0,C 180,E1 -7878.99,E2 -7878.99} C_VEL
LIN {X 0,Y 460.481,Z 229.611,A -85,B 0,C 180,E1 -7882.38,E2 -7882.38} C_VEL
LIN {X 0,Y 460.519,Z 229.617,A -85,B 0,C 180,E1 -7885.626,E2 -7885.626} C_VEL
LIN {X 0,Y 460.489,Z 229.62,A -85,B 0,C 180,E1 -7888.746,E2 -7888.746} C_VEL
LIN {X 0,Y 460.491,Z 229.61,A -85,B 0,C 180,E1 -7891.767,E2 -7891.767} C_VEL
LIN {X 0,Y 460.5,Z 229.616,A -85,B 0,C 180,E1 -7894.706,E2 -7894.706} C_VEL
LIN {X 0,Y 460.498,Z 229.624,A -85,B 0,C 180,E1 -7897.575,E2 -7897.575} C_VEL
LIN {X 0,Y 460.559,Z 229.603,A -85,B 0,C 180,E1 -7900.388,E2 -7900.388} C_VEL
LIN {X 0,Y 460.599,Z 229.602,A -85,B 0,C 180,E1 -7904.062,E2 -7904.062} C_VEL
LIN {X 0,Y 460.599,Z 229.611,A -85,B 0,C 180,E1 -7907.669,E2 -7907.669} C_VEL
LIN {X 0,Y 460.602,Z 229.602,A -85,B 0,C 180,E1 -7911.227,E2 -7911.227} C_VEL
LIN {X 0,Y 460.667,Z 229.587,A -85,B 0,C 180,E1 -7913.873,E2 -7913.873} C_VEL
LIN {X 0,Y 460.757,Z 229.582,A -85,B 0,C 180,E1 -7917.38,E2 -7917.38} C_VEL
LIN {X 0,Y 460.819,Z 229.584,A -85,B 0,C 180,E1 -7920.003,E2 -7920.003} C_VEL
LIN {X 0,Y 460.758,Z 229.582,A -85,B 0,C 180,E1 -7922.626,E2 -7922.626} C_VEL
LIN {X 0,Y 460.685,Z 229.584,A -85,B 0,C 180,E1 -7926.133,E2 -7926.133} C_VEL
LIN {X 0,Y 460.612,Z 229.608,A -85,B 0,C 180,E1 -7928.779,E2 -7928.779} C_VEL
LIN {X 0,Y 460.603,Z 229.611,A -85,B 0,C 180,E1 -7932.437,E2 -7932.437} C_VEL
LIN {X 0,Y 460.609,Z 229.594,A -85,B 0,C 180,E1 -7936,E2 -7936} C_VEL
LIN {X 0,Y 460.575,Z 229.609,A -85,B 0,C 180,E1 -7939.618,E2 -7939.618} C_VEL
LIN {X 0,Y 460.516,Z 229.616,A -85,B 0,C 180,E1 -7942.431,E2 -7942.431} C_VEL
LIN {X 0,Y 460.556,Z 229.609,A -85,B 0,C 180,E1 -7945.798,E2 -7945.798} C_VEL
LIN {X 0,Y 460.524,Z 229.616,A -85,B 0,C 180,E1 -7948.237,E2 -7948.237} C_VEL
LIN {X 0,Y 460.53,Z 229.614,A -85,B 0,C 180,E1 -7951.284,E2 -7951.284} C_VEL
LIN {X 0,Y 460.531,Z 229.615,A -85,B 0,C 180,E1 -7954.505,E2 -7954.505} C_VEL
LIN {X 0,Y 460.508,Z 229.619,A -85,B 0,C 180,E1 -7957.625,E2 -7957.625} C_VEL
LIN {X 0,Y 460.529,Z 229.617,A -85,B 0,C 180,E1 -7961.014,E2 -7961.014} C_VEL
LIN {X 0,Y 460.521,Z 229.616,A -85,B 0,C 180,E1 -7964.59,E2 -7964.59} C_VEL
LIN {X 0,Y 460.501,Z 229.626,A -85,B 0,C 180,E1 -7967.816,E2 -7967.816} C_VEL
LIN {X 0,Y 460.523,Z 229.621,A -85,B 0,C 180,E1 -7970.136,E2 -7970.136} C_VEL
LIN {X 0,Y 460.482,Z 229.625,A -85,B 0,C 180,E1 -7973.471,E2 -7973.471} C_VEL
LIN {X 0,Y 460.538,Z 229.614,A -85,B 0,C 180,E1 -7976.675,E2 -7976.675} C_VEL
LIN {X 0,Y 460.519,Z 229.619,A -85,B 0,C 180,E1 -7979.76,E2 -7979.76} C_VEL
LIN {X 0,Y 460.568,Z 229.614,A -85,B 0,C 180,E1 -7982.755,E2 -7982.755} C_VEL
LIN {X 0,Y 460.557,Z 229.65,A -85,B 0,C 180,E1 -7984.826,E2 -7984.826} C_VEL
LIN {X 0,Y 461.108,Z 232.34,A -85,B 0,C 180,E1 -7985.459,E2 -7985.459} C_VEL
LIN {X 0,Y 462.73,Z 242.061,A -85,B 0,C 180,E1 -7987.449,E2 -7987.449} C_VEL
LIN {X 0,Y 461.825,Z 260.689,A -85,B 0,C 180,E1 -7990.997,E2 -7990.997} C_VEL
LIN {X 0,Y 461.435,Z 269.989,A -85,B 0,C 180,E1 -7992.714,E2 -7992.714} C_VEL
LIN {X 0,Y 463.43,Z 282.062,A -85,B 0,C 180,E1 -7993.013,E2 -7993.013} C_VEL
LIN {X 0,Y 464.429,Z 289.288,A -85,B 0,C 180,E1 -7993.165,E2 -7993.165} C_VEL
LIN {X 0,Y 463.695,Z 377.425,A -85,B 0,C 180,E1 -7994.562,E2 -7994.562} C_VEL
LIN {X 0,Y 463.318,Z 390.777,A -85,B 0,C 180,E1 -7994.943,E2 -7994.943} C_VEL
LIN {X 0,Y 462.88,Z 403.548,A -85,B 0,C 180,E1 -7995.491,E2 -7995.491} C_VEL
LIN {X 0,Y 462.396,Z 414.894,A -85,B 0,C 180,E1 -7996.149,E2 -7996.149} C_VEL
LIN {X 0,Y 461.81,Z 426.973,A -85,B 0,C 180,E1 -7997.061,E2 -7997.061} C_VEL
LIN {X 0,Y 461.26,Z 438.152,A -85,B 0,C 180,E1 -7998.129,E2 -7998.129} C_VEL
LIN {X 0,Y 460.784,Z 447.374,A -85,B 0,C 180,E1 -7999.231,E2 -7999.231} C_VEL
LIN {X 0,Y 460.326,Z 456.343,A -85,B 0,C 180,E1 -8000.553,E2 -8000.553} C_VEL
LIN {X 0,Y 460.016,Z 463.564,A -85,B 0,C 180,E1 -8001.875,E2 -8001.875} C_VEL
LIN {X 0,Y 459.782,Z 468.434,A -85,B 0,C 180,E1 -8002.975,E2 -8002.975} C_VEL
LIN {X 0,Y 459.711,Z 473.168,A -85,B 0,C 180,E1 -8004.296,E2 -8004.296} C_VEL
LIN {X 0,Y 459.567,Z 476.783,A -85,B 0,C 180,E1 -8005.614,E2 -8005.614} C_VEL
LIN {X 0,Y 459.56,Z 478.649,A -85,B 0,C 180,E1 -8006.492,E2 -8006.492} C_VEL
LIN {X 0,Y 459.569,Z 480.05,A -85,B 0,C 180,E1 -8007.37,E2 -8007.37} C_VEL
LIN {X 0,Y 459.497,Z 481.655,A -85,B 0,C 180,E1 -8009.123,E2 -8009.123} C_VEL
LIN {X 0,Y 459.503,Z 481.875,A -85,B 0,C 180,E1 -8009.999,E2 -8009.999} C_VEL
LIN {X 0,Y 459.518,Z 481.055,A -85,B 0,C 180,E1 -8011.752,E2 -8011.752} C_VEL
LIN {X 0,Y 459.569,Z 480.062,A -85,B 0,C 180,E1 -8012.629,E2 -8012.629} C_VEL
LIN {X 0,Y 459.559,Z 478.669,A -85,B 0,C 180,E1 -8013.506,E2 -8013.506} C_VEL
LIN {X 0,Y 459.625,Z 475.738,A -85,B 0,C 180,E1 -8014.823,E2 -8014.823} C_VEL
LIN {X 0,Y 459.719,Z 470.744,A -85,B 0,C 180,E1 -8016.429,E2 -8016.429} C_VEL
LIN {X 0,Y 459.961,Z 464.655,A -85,B 0,C 180,E1 -8017.903,E2 -8017.903} C_VEL
LIN {X 0,Y 460.257,Z 457.759,A -85,B 0,C 180,E1 -8019.225,E2 -8019.225} C_VEL
LIN {X 0,Y 460.664,Z 449.13,A -85,B 0,C 180,E1 -8020.548,E2 -8020.548} C_VEL
LIN {X 0,Y 461.229,Z 440.281,A -85,B 0,C 180,E1 -8021.647,E2 -8021.647} C_VEL
LIN {X 0,Y 461.765,Z 430.434,A -85,B 0,C 180,E1 -8022.65,E2 -8022.65} C_VEL
LIN {X 0,Y 462.159,Z 419.937,A -85,B 0,C 180,E1 -8023.52,E2 -8023.52} C_VEL
LIN {X 0,Y 462.714,Z 408.058,A -85,B 0,C 180,E1 -8024.288,E2 -8024.288} C_VEL
LIN {X 0,Y 463.177,Z 395.703,A -85,B 0,C 180,E1 -8024.891,E2 -8024.891} C_VEL
LIN {X 0,Y 463.619,Z 383.02,A -85,B 0,C 180,E1 -8025.327,E2 -8025.327} C_VEL
LIN {X 0,Y 463.887,Z 367.977,A -85,B 0,C 180,E1 -8025.627,E2 -8025.627} C_VEL
LIN {X 0,Y 464.383,Z 287.569,A -85,B 0,C 180,E1 -8026.895,E2 -8026.895} C_VEL
LIN {X 0,Y 461.5,Z 270.264,A -85,B 0,C 180,E1 -8027.302,E2 -8027.302} C_VEL
LIN {X 0,Y 461.459,Z 268.512,A -85,B 0,C 180,E1 -8027.527,E2 -8027.527} C_VEL
LIN {X 0,Y 462.153,Z 251.534,A -85,B 0,C 180,E1 -8030.705,E2 -8030.705} C_VEL
LIN {X 0,Y 462.666,Z 241.763,A -85,B 0,C 180,E1 -8032.553,E2 -8032.553} C_VEL
LIN {X 0,Y 461.918,Z 236.377,A -85,B 0,C 180,E1 -8033.635,E2 -8033.635} C_VEL
LIN {X 0,Y 460.565,Z 229.731,A -85,B 0,C 180,E1 -8035.052,E2 -8035.052} C_VEL
LIN {X 0,Y 460.554,Z 229.617,A -85,B 0,C 180,E1 -8038.232,E2 -8038.232} C_VEL
LIN {X 0,Y 460.525,Z 229.62,A -85,B 0,C 180,E1 -8041.281,E2 -8041.281} C_VEL
LIN {X 0,Y 460.535,Z 229.618,A -85,B 0,C 180,E1 -8044.504,E2 -8044.504} C_VEL
LIN {X 0,Y 460.501,Z 229.619,A -85,B 0,C 180,E1 -8047.622,E2 -8047.622} C_VEL
LIN {X 0,Y 460.522,Z 229.615,A -85,B 0,C 180,E1 -8051.011,E2 -8051.011} C_VEL
LIN {X 0,Y 460.507,Z 229.624,A -85,B 0,C 180,E1 -8054.167,E2 -8054.167} C_VEL
LIN {X 0,Y 460.494,Z 229.621,A -85,B 0,C 180,E1 -8057.101,E2 -8057.101} C_VEL
LIN {X 0,Y 460.515,Z 229.622,A -85,B 0,C 180,E1 -8060.134,E2 -8060.134} C_VEL
LIN {X 0,Y 460.473,Z 229.622,A -85,B 0,C 180,E1 -8063.468,E2 -8063.468} C_VEL
LIN {X 0,Y 460.516,Z 229.624,A -85,B 0,C 180,E1 -8066.672,E2 -8066.672} C_VEL
LIN {X 0,Y 460.503,Z 229.618,A -85,B 0,C 180,E1 -8069.757,E2 -8069.757} C_VEL
LIN {X 0,Y 460.49,Z 229.623,A -85,B 0,C 180,E1 -8072.749,E2 -8072.749} C_VEL
LIN {X 0,Y 460.516,Z 229.616,A -85,B 0,C 180,E1 -8075.664,E2 -8075.664} C_VEL
LIN {X 0,Y 460.519,Z 229.618,A -85,B 0,C 180,E1 -8078.576,E2 -8078.576} C_VEL
LIN {X 0,Y 460.58,Z 229.608,A -85,B 0,C 180,E1 -8081.308,E2 -8081.308} C_VEL
LIN {X 0,Y 460.601,Z 229.606,A -85,B 0,C 180,E1 -8084.056,E2 -8084.056} C_VEL
LIN {X 0,Y 460.604,Z 229.608,A -85,B 0,C 180,E1 -8087.663,E2 -8087.663} C_VEL
LIN {X 0,Y 460.584,Z 229.61,A -85,B 0,C 180,E1 -8091.22,E2 -8091.22} C_VEL
LIN {X 0,Y 460.679,Z 229.599,A -85,B 0,C 180,E1 -8093.867,E2 -8093.867} C_VEL
LIN {X 0,Y 460.744,Z 229.59,A -85,B 0,C 180,E1 -8097.374,E2 -8097.374} C_VEL
LIN {X 0,Y 460.764,Z 229.585,A -85,B 0,C 180,E1 -8099.997,E2 -8099.997} C_VEL
LIN {X 0,Y 460.725,Z 229.59,A -85,B 0,C 180,E1 -8102.62,E2 -8102.62} C_VEL
LIN {X 0,Y 460.646,Z 229.603,A -85,B 0,C 180,E1 -8106.128,E2 -8106.128} C_VEL
LIN {X 0,Y 460.574,Z 229.609,A -85,B 0,C 180,E1 -8108.774,E2 -8108.774} C_VEL
LIN {X 0,Y 460.582,Z 229.61,A -85,B 0,C 180,E1 -8112.432,E2 -8112.432} C_VEL
LIN {X 0,Y 460.584,Z 229.615,A -85,B 0,C 180,E1 -8115.994,E2 -8115.994} C_VEL
LIN {X 0,Y 460.548,Z 229.616,A -85,B 0,C 180,E1 -8119.613,E2 -8119.613} C_VEL
LIN {X 0,Y 460.491,Z 229.624,A -85,B 0,C 180,E1 -8122.426,E2 -8122.426} C_VEL
LIN {X 0,Y 460.527,Z 229.617,A -85,B 0,C 180,E1 -8125.794,E2 -8125.794} C_VEL
LIN {X 0,Y 460.504,Z 229.62,A -85,B 0,C 180,E1 -8128.232,E2 -8128.232} C_VEL
LIN {X 0,Y 460.495,Z 229.62,A -85,B 0,C 180,E1 -8131.28,E2 -8131.28} C_VEL
LIN {X 0,Y 460.508,Z 229.623,A -85,B 0,C 180,E1 -8134.503,E2 -8134.503} C_VEL
LIN {X 0,Y 460.502,Z 229.619,A -85,B 0,C 180,E1 -8137.618,E2 -8137.618} C_VEL
LIN {X 0,Y 460.53,Z 229.621,A -85,B 0,C 180,E1 -8140.269,E2 -8140.269} C_VEL
LIN {X 0,Y 460.504,Z 229.625,A -85,B 0,C 180,E1 -8143.369,E2 -8143.369} C_VEL
LIN {X 0,Y 460.559,Z 229.805,A -85,B 0,C 180,E1 -8144.177,E2 -8144.177} C_VEL
LIN {X 0,Y 462.09,Z 238.053,A -85,B 0,C 180,E1 -8145.918,E2 -8145.918} C_VEL
LIN {X 0,Y 461.693,Z 251.531,A -85,B 0,C 180,E1 -8148.536,E2 -8148.536} C_VEL
LIN {X 0,Y 461.51,Z 257.896,A -85,B 0,C 180,E1 -8149.716,E2 -8149.716} C_VEL
LIN {X 0,Y 462.456,Z 263.011,A -85,B 0,C 180,E1 -8149.875,E2 -8149.875} C_VEL
LIN {X 0,Y 464.563,Z 276.017,A -85,B 0,C 180,E1 -8150.167,E2 -8150.167} C_VEL
LIN {X 0,Y 463.712,Z 366.016,A -85,B 0,C 180,E1 -8151.603,E2 -8151.603} C_VEL
LIN {X 0,Y 463.393,Z 379.034,A -85,B 0,C 180,E1 -8151.987,E2 -8151.987} C_VEL
LIN {X 0,Y 463.069,Z 391.264,A -85,B 0,C 180,E1 -8152.521,E2 -8152.521} C_VEL
LIN {X 0,Y 462.54,Z 403.626,A -85,B 0,C 180,E1 -8153.255,E2 -8153.255} C_VEL
LIN {X 0,Y 461.935,Z 415.206,A -85,B 0,C 180,E1 -8154.145,E2 -8154.145} C_VEL
LIN {X 0,Y 461.46,Z 424.543,A -85,B 0,C 180,E1 -8155.039,E2 -8155.039} C_VEL
LIN {X 0,Y 460.969,Z 434.325,A -85,B 0,C 180,E1 -8156.188,E2 -8156.188} C_VEL
LIN {X 0,Y 460.533,Z 442.523,A -85,B 0,C 180,E1 -8157.378,E2 -8157.378} C_VEL
LIN {X 0,Y 460.127,Z 450.379,A -85,B 0,C 180,E1 -8158.789,E2 -8158.789} C_VEL
LIN {X 0,Y 460.083,Z 451.747,A -85,B 0,C 180,E1 -8159.073,E2 -8159.073} C_VEL
LIN {X 0,Y 459.331,Z 454.647,A -85,B 0,C 180,E1 -8159.712,E2 -8159.712} C_VEL
LIN {X 0,Y 456.298,Z 458.9,A -85,B 0,C 180,E1 -8160.769,E2 -8160.769} C_VEL
LIN {X 0,Y 453.264,Z 462.429,A -85,B 0,C 180,E1 -8161.875,E2 -8161.875} C_VEL
LIN {X 0,Y 452.521,Z 464.215,A -85,B 0,C 180,E1 -8162.581,E2 -8162.581} C_VEL
LIN {X 0,Y 452.356,Z 467.361,A -85,B 0,C 180,E1 -8164.294,E2 -8164.294} C_VEL
LIN {X 0,Y 452.3,Z 468.382,A -85,B 0,C 180,E1 -8165.196,E2 -8165.196} C_VEL
LIN {X 0,Y 452.286,Z 469.149,A -85,B 0,C 180,E1 -8166.449,E2 -8166.449} C_VEL
LIN {X 0,Y 452.262,Z 468.93,A -85,B 0,C 180,E1 -8168.103,E2 -8168.103} C_VEL
LIN {X 0,Y 452.34,Z 468.195,A -85,B 0,C 180,E1 -8169.063,E2 -8169.063} C_VEL
LIN {X 0,Y 452.371,Z 466.991,A -85,B 0,C 180,E1 -8170.015,E2 -8170.015} C_VEL
LIN {X 0,Y 452.515,Z 464.585,A -85,B 0,C 180,E1 -8171.317,E2 -8171.317} C_VEL
LIN {X 0,Y 452.643,Z 460.533,A -85,B 0,C 180,E1 -8172.843,E2 -8172.843} C_VEL
LIN {X 0,Y 452.917,Z 454.74,A -85,B 0,C 180,E1 -8174.447,E2 -8174.447} C_VEL
LIN {X 0,Y 453.218,Z 448.126,A -85,B 0,C 180,E1 -8175.864,E2 -8175.864} C_VEL
LIN {X 0,Y 453.648,Z 439.799,A -85,B 0,C 180,E1 -8177.27,E2 -8177.27} C_VEL
LIN {X 0,Y 454.112,Z 431.604,A -85,B 0,C 180,E1 -8178.394,E2 -8178.394} C_VEL
LIN {X 0,Y 454.649,Z 421.426,A -85,B 0,C 180,E1 -8179.536,E2 -8179.536} C_VEL
LIN {X 0,Y 455.222,Z 411.251,A -85,B 0,C 180,E1 -8180.45,E2 -8180.45} C_VEL
LIN {X 0,Y 455.761,Z 400.232,A -85,B 0,C 180,E1 -8181.242,E2 -8181.242} C_VEL
LIN {X 0,Y 456.217,Z 388.071,A -85,B 0,C 180,E1 -8181.92,E2 -8181.92} C_VEL
LIN {X 0,Y 456.564,Z 375.582,A -85,B 0,C 180,E1 -8182.427,E2 -8182.427} C_VEL
LIN {X 0,Y 456.906,Z 362.313,A -85,B 0,C 180,E1 -8182.766,E2 -8182.766} C_VEL
LIN {X 0,Y 457.525,Z 274.481,A -85,B 0,C 180,E1 -8184.174,E2 -8184.174} C_VEL
LIN {X 0,Y 454.611,Z 258.462,A -85,B 0,C 180,E1 -8184.567,E2 -8184.567} C_VEL
LIN {X 0,Y 454.663,Z 255.41,A -85,B 0,C 180,E1 -8185.124,E2 -8185.124} C_VEL
LIN {X 0,Y 455.321,Z 241.552,A -85,B 0,C 180,E1 -8188.011,E2 -8188.011} C_VEL
LIN {X 0,Y 454.111,Z 232.513,A -85,B 0,C 180,E1 -8190.001,E2 -8190.001} C_VEL
LIN {X 0,Y 453.757,Z 230.492,A -85,B 0,C 180,E1 -8190.528,E2 -8190.528} C_VEL
LIN {X 0,Y 453.729,Z 230.467,A -85,B 0,C 180,E1 -8192.664,E2 -8192.664} C_VEL
LIN {X 0,Y 453.638,Z 230.475,A -85,B 0,C 180,E1 -8196.227,E2 -8196.227} C_VEL
LIN {X 0,Y 453.555,Z 230.486,A -85,B 0,C 180,E1 -8198.915,E2 -8198.915} C_VEL
LIN {X 0,Y 453.566,Z 230.477,A -85,B 0,C 180,E1 -8202.552,E2 -8202.552} C_VEL
LIN {X 0,Y 453.51,Z 230.491,A -85,B 0,C 180,E1 -8206.198,E2 -8206.198} C_VEL
LIN {X 0,Y 453.485,Z 230.492,A -85,B 0,C 180,E1 -8209.042,E2 -8209.042} C_VEL
LIN {X 0,Y 453.442,Z 230.504,A -85,B 0,C 180,E1 -8211.838,E2 -8211.838} C_VEL
LIN {X 0,Y 453.467,Z 230.494,A -85,B 0,C 180,E1 -8214.738,E2 -8214.738} C_VEL
LIN {X 0,Y 453.474,Z 230.499,A -85,B 0,C 180,E1 -8217.956,E2 -8217.956} C_VEL
LIN {X 0,Y 453.445,Z 230.499,A -85,B 0,C 180,E1 -8220.762,E2 -8220.762} C_VEL
LIN {X 0,Y 453.437,Z 230.5,A -85,B 0,C 180,E1 -8223.917,E2 -8223.917} C_VEL
LIN {X 0,Y 453.411,Z 230.502,A -85,B 0,C 180,E1 -8227.194,E2 -8227.194} C_VEL
LIN {X 0,Y 453.444,Z 230.5,A -85,B 0,C 180,E1 -8230.615,E2 -8230.615} C_VEL
LIN {X 0,Y 453.434,Z 230.495,A -85,B 0,C 180,E1 -8234.225,E2 -8234.225} C_VEL
LIN {X 0,Y 453.4,Z 230.508,A -85,B 0,C 180,E1 -8237.004,E2 -8237.004} C_VEL
LIN {X 0,Y 453.45,Z 230.491,A -85,B 0,C 180,E1 -8239.416,E2 -8239.416} C_VEL
LIN {X 0,Y 453.433,Z 230.494,A -85,B 0,C 180,E1 -8242.814,E2 -8242.814} C_VEL
LIN {X 0,Y 453.45,Z 230.496,A -85,B 0,C 180,E1 -8246.09,E2 -8246.09} C_VEL
LIN {X 0,Y 453.44,Z 230.495,A -85,B 0,C 180,E1 -8249.242,E2 -8249.242} C_VEL
LIN {X 0,Y 453.459,Z 230.483,A -85,B 0,C 180,E1 -8252.297,E2 -8252.297} C_VEL
LIN {X 0,Y 453.453,Z 230.499,A -85,B 0,C 180,E1 -8255.266,E2 -8255.266} C_VEL
LIN {X 0,Y 453.472,Z 230.492,A -85,B 0,C 180,E1 -8258.419,E2 -8258.419} C_VEL
LIN {X 0,Y 453.515,Z 230.481,A -85,B 0,C 180,E1 -8261.012,E2 -8261.012} C_VEL
LIN {X 0,Y 453.564,Z 230.477,A -85,B 0,C 180,E1 -8263.883,E2 -8263.883} C_VEL
LIN {X 0,Y 453.561,Z 230.485,A -85,B 0,C 180,E1 -8267.475,E2 -8267.475} C_VEL
LIN {X 0,Y 453.568,Z 230.478,A -85,B 0,C 180,E1 -8271.09,E2 -8271.09} C_VEL
LIN {X 0,Y 453.635,Z 230.462,A -85,B 0,C 180,E1 -8273.777,E2 -8273.777} C_VEL
LIN {X 0,Y 453.704,Z 230.46,A -85,B 0,C 180,E1 -8277.34,E2 -8277.34} C_VEL
LIN {X 0,Y 453.768,Z 230.462,A -85,B 0,C 180,E1 -8280.003,E2 -8280.003} C_VEL
LIN {X 0,Y 453.704,Z 230.46,A -85,B 0,C 180,E1 -8282.666,E2 -8282.666} C_VEL
LIN {X 0,Y 453.654,Z 230.461,A -85,B 0,C 180,E1 -8286.228,E2 -8286.228} C_VEL
LIN {X 0,Y 453.577,Z 230.483,A -85,B 0,C 180,E1 -8288.916,E2 -8288.916} C_VEL
LIN {X 0,Y 453.571,Z 230.485,A -85,B 0,C 180,E1 -8292.531,E2 -8292.531} C_VEL
LIN {X 0,Y 453.552,Z 230.474,A -85,B 0,C 180,E1 -8296.198,E2 -8296.198} C_VEL
LIN {X 0,Y 453.525,Z 230.493,A -85,B 0,C 180,E1 -8299.041,E2 -8299.041} C_VEL
LIN {X 0,Y 453.484,Z 230.49,A -85,B 0,C 180,E1 -8301.838,E2 -8301.838} C_VEL
LIN {X 0,Y 453.503,Z 230.483,A -85,B 0,C 180,E1 -8304.737,E2 -8304.737} C_VEL
LIN {X 0,Y 453.485,Z 230.493,A -85,B 0,C 180,E1 -8307.948,E2 -8307.948} C_VEL
LIN {X 0,Y 453.484,Z 230.492,A -85,B 0,C 180,E1 -8310.761,E2 -8310.761} C_VEL
LIN {X 0,Y 453.476,Z 230.495,A -85,B 0,C 180,E1 -8313.915,E2 -8313.915} C_VEL
LIN {X 0,Y 453.459,Z 230.497,A -85,B 0,C 180,E1 -8317.191,E2 -8317.191} C_VEL
LIN {X 0,Y 453.481,Z 230.493,A -85,B 0,C 180,E1 -8320.613,E2 -8320.613} C_VEL
LIN {X 0,Y 453.469,Z 230.496,A -85,B 0,C 180,E1 -8324.223,E2 -8324.223} C_VEL
LIN {X 0,Y 453.447,Z 230.496,A -85,B 0,C 180,E1 -8327.003,E2 -8327.003} C_VEL
LIN {X 0,Y 453.481,Z 230.497,A -85,B 0,C 180,E1 -8329.413,E2 -8329.413} C_VEL
LIN {X 0,Y 453.459,Z 230.497,A -85,B 0,C 180,E1 -8332.81,E2 -8332.81} C_VEL
LIN {X 0,Y 453.486,Z 230.495,A -85,B 0,C 180,E1 -8336.088,E2 -8336.088} C_VEL
LIN {X 0,Y 453.486,Z 230.493,A -85,B 0,C 180,E1 -8339.241,E2 -8339.241} C_VEL
LIN {X 0,Y 453.542,Z 230.492,A -85,B 0,C 180,E1 -8342.297,E2 -8342.297} C_VEL
LIN {X 0,Y 453.553,Z 230.605,A -85,B 0,C 180,E1 -8344.655,E2 -8344.655} C_VEL
LIN {X 0,Y 455.466,Z 240.717,A -85,B 0,C 180,E1 -8346.829,E2 -8346.829} C_VEL
LIN {X 0,Y 455.768,Z 244.533,A -85,B 0,C 180,E1 -8347.598,E2 -8347.598} C_VEL
LIN {X 0,Y 454.795,Z 262.477,A -85,B 0,C 180,E1 -8351.063,E2 -8351.063} C_VEL
LIN {X 0,Y 454.474,Z 269.907,A -85,B 0,C 180,E1 -8352.45,E2 -8352.45} C_VEL
LIN {X 0,Y 457.071,Z 285.585,A -85,B 0,C 180,E1 -8352.835,E2 -8352.835} C_VEL
LIN {X 0,Y 457.652,Z 291.739,A -85,B 0,C 180,E1 -8352.956,E2 -8352.956} C_VEL
LIN {X 0,Y 456.813,Z 378.246,A -85,B 0,C 180,E1 -8354.352,E2 -8354.352} C_VEL
LIN {X 0,Y 456.44,Z 392.049,A -85,B 0,C 180,E1 -8354.768,E2 -8354.768} C_VEL
LIN {X 0,Y 455.961,Z 404.438,A -85,B 0,C 180,E1 -8355.323,E2 -8355.323} C_VEL
LIN {X 0,Y 455.404,Z 416.304,A -85,B 0,C 180,E1 -8356.046,E2 -8356.046} C_VEL
LIN {X 0,Y 454.828,Z 427.695,A -85,B 0,C 180,E1 -8356.937,E2 -8356.937} C_VEL
LIN {X 0,Y 454.308,Z 438.003,A -85,B 0,C 180,E1 -8357.945,E2 -8357.945} C_VEL
LIN {X 0,Y 453.78,Z 447.236,A -85,B 0,C 180,E1 -8359.063,E2 -8359.063} C_VEL
LIN {X 0,Y 453.29,Z 456.213,A -85,B 0,C 180,E1 -8360.405,E2 -8360.405} C_VEL
LIN {X 0,Y 452.949,Z 463.44,A -85,B 0,C 180,E1 -8361.748,E2 -8361.748} C_VEL
LIN {X 0,Y 452.728,Z 468.316,A -85,B 0,C 180,E1 -8362.865,E2 -8362.865} C_VEL
LIN {X 0,Y 452.611,Z 473.054,A -85,B 0,C 180,E1 -8364.207,E2 -8364.207} C_VEL
LIN {X 0,Y 452.49,Z 476.674,A -85,B 0,C 180,E1 -8365.545,E2 -8365.545} C_VEL
LIN {X 0,Y 452.458,Z 478.543,A -85,B 0,C 180,E1 -8366.437,E2 -8366.437} C_VEL
LIN {X 0,Y 452.493,Z 479.946,A -85,B 0,C 180,E1 -8367.329,E2 -8367.329} C_VEL
LIN {X 0,Y 452.406,Z 481.555,A -85,B 0,C 180,E1 -8369.109,E2 -8369.109} C_VEL
LIN {X 0,Y 452.409,Z 481.776,A -85,B 0,C 180,E1 -8369.999,E2 -8369.999} C_VEL
LIN {X 0,Y 452.435,Z 480.96,A -85,B 0,C 180,E1 -8371.78,E2 -8371.78} C_VEL
LIN {X 0,Y 452.493,Z 479.968,A -85,B 0,C 180,E1 -8372.67,E2 -8372.67} C_VEL
LIN {X 0,Y 452.457,Z 478.576,A -85,B 0,C 180,E1 -8373.561,E2 -8373.561} C_VEL
LIN {X 0,Y 452.557,Z 475.646,A -85,B 0,C 180,E1 -8374.899,E2 -8374.899} C_VEL
LIN {X 0,Y 452.635,Z 471.071,A -85,B 0,C 180,E1 -8376.415,E2 -8376.415} C_VEL
LIN {X 0,Y 452.902,Z 464.567,A -85,B 0,C 180,E1 -8378.027,E2 -8378.027} C_VEL
LIN {X 0,Y 453.232,Z 457.672,A -85,B 0,C 180,E1 -8379.37,E2 -8379.37} C_VEL
LIN {X 0,Y 453.595,Z 450.633,A -85,B 0,C 180,E1 -8380.489,E2 -8380.489} C_VEL
LIN {X 0,Y 454.109,Z 442.15,A -85,B 0,C 180,E1 -8381.606,E2 -8381.606} C_VEL
LIN {X 0,Y 454.736,Z 432.38,A -85,B 0,C 180,E1 -8382.653,E2 -8382.653} C_VEL
LIN {X 0,Y 455.155,Z 421.293,A -85,B 0,C 180,E1 -8383.619,E2 -8383.619} C_VEL
LIN {X 0,Y 455.748,Z 409.93,A -85,B 0,C 180,E1 -8384.397,E2 -8384.397} C_VEL
LIN {X 0,Y 456.216,Z 398.273,A -85,B 0,C 180,E1 -8385.01,E2 -8385.01} C_VEL
LIN {X 0,Y 456.737,Z 384.861,A -85,B 0,C 180,E1 -8385.506,E2 -8385.506} C_VEL
LIN {X 0,Y 457.011,Z 371.655,A -85,B 0,C 180,E1 -8385.811,E2 -8385.811} C_VEL
LIN {X 0,Y 457.597,Z 288.567,A -85,B 0,C 180,E1 -8387.14,E2 -8387.14} C_VEL
LIN {X 0,Y 454.493,Z 269.904,A -85,B 0,C 180,E1 -8387.595,E2 -8387.595} C_VEL
LIN {X 0,Y 454.613,Z 266.132,A -85,B 0,C 180,E1 -8388.242,E2 -8388.242} C_VEL
LIN {X 0,Y 455.4,Z 249.014,A -85,B 0,C 180,E1 -8391.5,E2 -8391.5} C_VEL
LIN {X 0,Y 455.67,Z 241.685,A -85,B 0,C 180,E1 -8392.919,E2 -8392.919} C_VEL
LIN {X 0,Y 453.526,Z 230.589,A -85,B 0,C 180,E1 -8395.284,E2 -8395.284} C_VEL
LIN {X 0,Y 453.512,Z 230.493,A -85,B 0,C 180,E1 -8398.711,E2 -8398.711} C_VEL
LIN {X 0,Y 453.468,Z 230.499,A -85,B 0,C 180,E1 -8401.798,E2 -8401.798} C_VEL
LIN {X 0,Y 453.483,Z 230.495,A -85,B 0,C 180,E1 -8404.988,E2 -8404.988} C_VEL
LIN {X 0,Y 453.46,Z 230.501,A -85,B 0,C 180,E1 -8408.311,E2 -8408.311} C_VEL
LIN {X 0,Y 453.474,Z 230.496,A -85,B 0,C 180,E1 -8410.61,E2 -8410.61} C_VEL
LIN {X 0,Y 453.462,Z 230.502,A -85,B 0,C 180,E1 -8414.22,E2 -8414.22} C_VEL
LIN {X 0,Y 453.45,Z 230.499,A -85,B 0,C 180,E1 -8417.001,E2 -8417.001} C_VEL
LIN {X 0,Y 453.473,Z 230.494,A -85,B 0,C 180,E1 -8419.411,E2 -8419.411} C_VEL
LIN {X 0,Y 453.45,Z 230.502,A -85,B 0,C 180,E1 -8422.808,E2 -8422.808} C_VEL
LIN {X 0,Y 453.467,Z 230.496,A -85,B 0,C 180,E1 -8426.084,E2 -8426.084} C_VEL
LIN {X 0,Y 453.474,Z 230.495,A -85,B 0,C 180,E1 -8429.238,E2 -8429.238} C_VEL
LIN {X 0,Y 453.473,Z 230.495,A -85,B 0,C 180,E1 -8432.291,E2 -8432.291} C_VEL
LIN {X 0,Y 453.468,Z 230.497,A -85,B 0,C 180,E1 -8435.26,E2 -8435.26} C_VEL
LIN {X 0,Y 453.478,Z 230.493,A -85,B 0,C 180,E1 -8438.413,E2 -8438.413} C_VEL
LIN {X 0,Y 453.52,Z 230.49,A -85,B 0,C 180,E1 -8441.006,E2 -8441.006} C_VEL
LIN {X 0,Y 453.566,Z 230.483,A -85,B 0,C 180,E1 -8443.877,E2 -8443.877} C_VEL
LIN {X 0,Y 453.56,Z 230.487,A -85,B 0,C 180,E1 -8447.468,E2 -8447.468} C_VEL
LIN {X 0,Y 453.554,Z 230.486,A -85,B 0,C 180,E1 -8451.083,E2 -8451.083} C_VEL
LIN {X 0,Y 453.647,Z 230.476,A -85,B 0,C 180,E1 -8453.771,E2 -8453.771} C_VEL
LIN {X 0,Y 453.691,Z 230.467,A -85,B 0,C 180,E1 -8457.333,E2 -8457.333} C_VEL
LIN {X 0,Y 453.715,Z 230.463,A -85,B 0,C 180,E1 -8459.997,E2 -8459.997} C_VEL
LIN {X 0,Y 453.674,Z 230.468,A -85,B 0,C 180,E1 -8462.661,E2 -8462.661} C_VEL
LIN {X 0,Y 453.614,Z 230.478,A -85,B 0,C 180,E1 -8466.223,E2 -8466.223} C_VEL
LIN {X 0,Y 453.544,Z 230.484,A -85,B 0,C 180,E1 -8468.911,E2 -8468.911} C_VEL
LIN {X 0,Y 453.549,Z 230.485,A -85,B 0,C 180,E1 -8472.526,E2 -8472.526} C_VEL
LIN {X 0,Y 453.527,Z 230.491,A -85,B 0,C 180,E1 -8476.193,E2 -8476.193} C_VEL
LIN {X 0,Y 453.498,Z 230.492,A -85,B 0,C 180,E1 -8479.036,E2 -8479.036} C_VEL
LIN {X 0,Y 453.457,Z 230.501,A -85,B 0,C 180,E1 -8481.833,E2 -8481.833} C_VEL
LIN {X 0,Y 453.479,Z 230.495,A -85,B 0,C 180,E1 -8484.732,E2 -8484.732} C_VEL
LIN {X 0,Y 453.484,Z 230.497,A -85,B 0,C 180,E1 -8487.95,E2 -8487.95} C_VEL
LIN {X 0,Y 453.451,Z 230.501,A -85,B 0,C 180,E1 -8490.757,E2 -8490.757} C_VEL
LIN {X 0,Y 453.453,Z 230.5,A -85,B 0,C 180,E1 -8493.91,E2 -8493.91} C_VEL
LIN {X 0,Y 453.444,Z 230.499,A -85,B 0,C 180,E1 -8497.185,E2 -8497.185} C_VEL
LIN {X 0,Y 453.503,Z 230.494,A -85,B 0,C 180,E1 -8499.443,E2 -8499.443} C_VEL
LIN {X 0,Y 453.468,Z 230.501,A -85,B 0,C 180,E1 -8502.988,E2 -8502.988} C_VEL
LIN {X 0,Y 453.522,Z 230.645,A -85,B 0,C 180,E1 -8503.946,E2 -8503.946} C_VEL
LIN {X 0,Y 455.026,Z 238.465,A -85,B 0,C 180,E1 -8505.636,E2 -8505.636} C_VEL
LIN {X 0,Y 454.964,Z 246.245,A -85,B 0,C 180,E1 -8507.182,E2 -8507.182} C_VEL
LIN {X 0,Y 454.531,Z 257.9,A -85,B 0,C 180,E1 -8509.423,E2 -8509.423} C_VEL
LIN {X 0,Y 455.25,Z 261.742,A -85,B 0,C 180,E1 -8509.566,E2 -8509.566} C_VEL
LIN {X 0,Y 457.783,Z 275.714,A -85,B 0,C 180,E1 -8509.897,E2 -8509.897} C_VEL
LIN {X 0,Y 456.904,Z 365.57,A -85,B 0,C 180,E1 -8511.349,E2 -8511.349} C_VEL
LIN {X 0,Y 456.56,Z 379.022,A -85,B 0,C 180,E1 -8511.748,E2 -8511.748} C_VEL
LIN {X 0,Y 456.197,Z 391.668,A -85,B 0,C 180,E1 -8512.31,E2 -8512.31} C_VEL
LIN {X 0,Y 455.67,Z 403.497,A -85,B 0,C 180,E1 -8513.023,E2 -8513.023} C_VEL
LIN {X 0,Y 455.002,Z 415.29,A -85,B 0,C 180,E1 -8513.941,E2 -8513.941} C_VEL
LIN {X 0,Y 454.506,Z 424.473,A -85,B 0,C 180,E1 -8514.832,E2 -8514.832} C_VEL
LIN {X 0,Y 454.029,Z 433.288,A -85,B 0,C 180,E1 -8515.868,E2 -8515.868} C_VEL
LIN {X 0,Y 453.534,Z 442.216,A -85,B 0,C 180,E1 -8517.157,E2 -8517.157} C_VEL
LIN {X 0,Y 453.103,Z 449.901,A -85,B 0,C 180,E1 -8518.541,E2 -8518.541} C_VEL
LIN {X 0,Y 452.925,Z 455.184,A -85,B 0,C 180,E1 -8519.716,E2 -8519.716} C_VEL
LIN {X 0,Y 452.638,Z 460.588,A -85,B 0,C 180,E1 -8521.229,E2 -8521.229} C_VEL
LIN {X 0,Y 452.521,Z 464.215,A -85,B 0,C 180,E1 -8522.581,E2 -8522.581} C_VEL
LIN {X 0,Y 451.79,Z 465.787,A -85,B 0,C 180,E1 -8523.296,E2 -8523.296} C_VEL
LIN {X 0,Y 448.822,Z 467.766,A -85,B 0,C 180,E1 -8524.474,E2 -8524.474} C_VEL
LIN {X 0,Y 446.335,Z 468.766,A -85,B 0,C 180,E1 -8525.436,E2 -8525.436} C_VEL
LIN {X 0,Y 445.264,Z 469.174,A -85,B 0,C 180,E1 -8526.185,E2 -8526.185} C_VEL
LIN {X 0,Y 445.175,Z 469.242,A -85,B 0,C 180,E1 -8526.44,E2 -8526.44} C_VEL
LIN {X 0,Y 445.168,Z 469.22,A -85,B 0,C 180,E1 -8527.736,E2 -8527.736} C_VEL
LIN {X 0,Y 445.205,Z 468.63,A -85,B 0,C 180,E1 -8528.712,E2 -8528.712} C_VEL
LIN {X 0,Y 445.249,Z 467.602,A -85,B 0,C 180,E1 -8529.681,E2 -8529.681} C_VEL
LIN {X 0,Y 445.41,Z 465.055,A -85,B 0,C 180,E1 -8531.198,E2 -8531.198} C_VEL
LIN {X 0,Y 445.516,Z 461.719,A -85,B 0,C 180,E1 -8532.56,E2 -8532.56} C_VEL
LIN {X 0,Y 445.743,Z 456.702,A -85,B 0,C 180,E1 -8534.091,E2 -8534.091} C_VEL
LIN {X 0,Y 446.073,Z 450.032,A -85,B 0,C 180,E1 -8535.633,E2 -8535.633} C_VEL
LIN {X 0,Y 446.477,Z 442.357,A -85,B 0,C 180,E1 -8537.039,E2 -8537.039} C_VEL
LIN {X 0,Y 446.955,Z 434.501,A -85,B 0,C 180,E1 -8538.206,E2 -8538.206} C_VEL
LIN {X 0,Y 447.471,Z 424.934,A -85,B 0,C 180,E1 -8539.366,E2 -8539.366} C_VEL
LIN {X 0,Y 448.106,Z 414.23,A -85,B 0,C 180,E1 -8540.409,E2 -8540.409} C_VEL
LIN {X 0,Y 448.688,Z 403.913,A -85,B 0,C 180,E1 -8541.216,E2 -8541.216} C_VEL
LIN {X 0,Y 449.212,Z 391.797,A -85,B 0,C 180,E1 -8541.963,E2 -8541.963} C_VEL
LIN {X 0,Y 449.635,Z 379.052,A -85,B 0,C 180,E1 -8542.535,E2 -8542.535} C_VEL
LIN {X 0,Y 449.986,Z 365.749,A -85,B 0,C 180,E1 -8542.936,E2 -8542.936} C_VEL
LIN {X 0,Y 450.813,Z 275.819,A -85,B 0,C 180,E1 -8544.409,E2 -8544.409} C_VEL
LIN {X 0,Y 447.655,Z 258.416,A -85,B 0,C 180,E1 -8544.85,E2 -8544.85} C_VEL
LIN {X 0,Y 447.889,Z 251.862,A -85,B 0,C 180,E1 -8546.177,E2 -8546.177} C_VEL
LIN {X 0,Y 448.336,Z 242.288,A -85,B 0,C 180,E1 -8548.204,E2 -8548.204} C_VEL
LIN {X 0,Y 446.905,Z 232.287,A -85,B 0,C 180,E1 -8550.451,E2 -8550.451} C_VEL
LIN {X 0,Y 446.707,Z 231.368,A -85,B 0,C 180,E1 -8550.733,E2 -8550.733} C_VEL
LIN {X 0,Y 446.673,Z 231.346,A -85,B 0,C 180,E1 -8552.706,E2 -8552.706} C_VEL
LIN {X 0,Y 446.606,Z 231.35,A -85,B 0,C 180,E1 -8556.325,E2 -8556.325} C_VEL
LIN {X 0,Y 446.501,Z 231.366,A -85,B 0,C 180,E1 -8559.057,E2 -8559.057} C_VEL
LIN {X 0,Y 446.498,Z 231.357,A -85,B 0,C 180,E1 -8562.731,E2 -8562.731} C_VEL
LIN {X 0,Y 446.455,Z 231.368,A -85,B 0,C 180,E1 -8566.461,E2 -8566.461} C_VEL
LIN {X 0,Y 446.435,Z 231.372,A -85,B 0,C 180,E1 -8569.305,E2 -8569.305} C_VEL
LIN {X 0,Y 446.384,Z 231.382,A -85,B 0,C 180,E1 -8572.202,E2 -8572.202} C_VEL
LIN {X 0,Y 446.409,Z 231.372,A -85,B 0,C 180,E1 -8575.156,E2 -8575.156} C_VEL
LIN {X 0,Y 446.417,Z 231.375,A -85,B 0,C 180,E1 -8578.184,E2 -8578.184} C_VEL
LIN {X 0,Y 446.384,Z 231.377,A -85,B 0,C 180,E1 -8581.303,E2 -8581.303} C_VEL
LIN {X 0,Y 446.392,Z 231.373,A -85,B 0,C 180,E1 -8584.527,E2 -8584.527} C_VEL
LIN {X 0,Y 446.374,Z 231.38,A -85,B 0,C 180,E1 -8588.08,E2 -8588.08} C_VEL
LIN {X 0,Y 446.376,Z 231.372,A -85,B 0,C 180,E1 -8591.398,E2 -8591.398} C_VEL
LIN {X 0,Y 446.426,Z 231.375,A -85,B 0,C 180,E1 -8595.108,E2 -8595.108} C_VEL
LIN {X 0,Y 446.379,Z 231.382,A -85,B 0,C 180,E1 -8598.609,E2 -8598.609} C_VEL
LIN {X 0,Y 446.392,Z 231.364,A -85,B 0,C 180,E1 -8601.925,E2 -8601.925} C_VEL
LIN {X 0,Y 446.405,Z 231.377,A -85,B 0,C 180,E1 -8605.48,E2 -8605.48} C_VEL
LIN {X 0,Y 446.392,Z 231.375,A -85,B 0,C 180,E1 -8608.703,E2 -8608.703} C_VEL
LIN {X 0,Y 446.41,Z 231.362,A -85,B 0,C 180,E1 -8611.84,E2 -8611.84} C_VEL
LIN {X 0,Y 446.403,Z 231.373,A -85,B 0,C 180,E1 -8614.849,E2 -8614.849} C_VEL
LIN {X 0,Y 446.439,Z 231.368,A -85,B 0,C 180,E1 -8618.249,E2 -8618.249} C_VEL
LIN {X 0,Y 446.441,Z 231.357,A -85,B 0,C 180,E1 -8621.652,E2 -8621.652} C_VEL
LIN {X 0,Y 446.5,Z 231.354,A -85,B 0,C 180,E1 -8624.483,E2 -8624.483} C_VEL
LIN {X 0,Y 446.503,Z 231.365,A -85,B 0,C 180,E1 -8628.196,E2 -8628.196} C_VEL
LIN {X 0,Y 446.515,Z 231.356,A -85,B 0,C 180,E1 -8630.948,E2 -8630.948} C_VEL
LIN {X 0,Y 446.605,Z 231.337,A -85,B 0,C 180,E1 -8633.679,E2 -8633.679} C_VEL
LIN {X 0,Y 446.654,Z 231.338,A -85,B 0,C 180,E1 -8637.298,E2 -8637.298} C_VEL
LIN {X 0,Y 446.718,Z 231.34,A -85,B 0,C 180,E1 -8640.003,E2 -8640.003} C_VEL
LIN {X 0,Y 446.654,Z 231.337,A -85,B 0,C 180,E1 -8642.709,E2 -8642.709} C_VEL
LIN {X 0,Y 446.625,Z 231.337,A -85,B 0,C 180,E1 -8646.327,E2 -8646.327} C_VEL
LIN {X 0,Y 446.525,Z 231.36,A -85,B 0,C 180,E1 -8649.058,E2 -8649.058} C_VEL
LIN {X 0,Y 446.528,Z 231.359,A -85,B 0,C 180,E1 -8652.732,E2 -8652.732} C_VEL
LIN {X 0,Y 446.496,Z 231.355,A -85,B 0,C 180,E1 -8656.461,E2 -8656.461} C_VEL
LIN {X 0,Y 446.477,Z 231.368,A -85,B 0,C 180,E1 -8659.305,E2 -8659.305} C_VEL
LIN {X 0,Y 446.425,Z 231.37,A -85,B 0,C 180,E1 -8662.202,E2 -8662.202} C_VEL
LIN {X 0,Y 446.447,Z 231.368,A -85,B 0,C 180,E1 -8665.155,E2 -8665.155} C_VEL
LIN {X 0,Y 446.448,Z 231.369,A -85,B 0,C 180,E1 -8668.184,E2 -8668.184} C_VEL
LIN {X 0,Y 446.424,Z 231.37,A -85,B 0,C 180,E1 -8671.302,E2 -8671.302} C_VEL
LIN {X 0,Y 446.431,Z 231.372,A -85,B 0,C 180,E1 -8674.525,E2 -8674.525} C_VEL
LIN {X 0,Y 446.42,Z 231.371,A -85,B 0,C 180,E1 -8678.079,E2 -8678.079} C_VEL
LIN {X 0,Y 446.417,Z 231.378,A -85,B 0,C 180,E1 -8681.395,E2 -8681.395} C_VEL
LIN {X 0,Y 446.432,Z 231.372,A -85,B 0,C 180,E1 -8684.893,E2 -8684.893} C_VEL
LIN {X 0,Y 446.402,Z 231.382,A -85,B 0,C 180,E1 -8687.73,E2 -8687.73} C_VEL
LIN {X 0,Y 446.417,Z 231.374,A -85,B 0,C 180,E1 -8690.97,E2 -8690.97} C_VEL
LIN {X 0,Y 446.428,Z 231.376,A -85,B 0,C 180,E1 -8694.374,E2 -8694.374} C_VEL
LIN {X 0,Y 446.432,Z 231.374,A -85,B 0,C 180,E1 -8697.639,E2 -8697.639} C_VEL
LIN {X 0,Y 446.456,Z 231.371,A -85,B 0,C 180,E1 -8700.791,E2 -8700.791} C_VEL
LIN {X 0,Y 446.454,Z 231.373,A -85,B 0,C 180,E1 -8703.846,E2 -8703.846} C_VEL
LIN {X 0,Y 446.51,Z 231.585,A -85,B 0,C 180,E1 -8704.476,E2 -8704.476} C_VEL
LIN {X 0,Y 448.656,Z 243.019,A -85,B 0,C 180,E1 -8706.944,E2 -8706.944} C_VEL
LIN {X 0,Y 448.729,Z 246.519,A -85,B 0,C 180,E1 -8707.651,E2 -8707.651} C_VEL
LIN {X 0,Y 447.803,Z 263.546,A -85,B 0,C 180,E1 -8710.994,E2 -8710.994} C_VEL
LIN {X 0,Y 447.535,Z 269.862,A -85,B 0,C 180,E1 -8712.181,E2 -8712.181} C_VEL
LIN {X 0,Y 450.841,Z 290.374,A -85,B 0,C 180,E1 -8712.678,E2 -8712.678} C_VEL
LIN {X 0,Y 449.979,Z 377.855,A -85,B 0,C 180,E1 -8714.108,E2 -8714.108} C_VEL
LIN {X 0,Y 449.556,Z 391.756,A -85,B 0,C 180,E1 -8714.529,E2 -8714.529} C_VEL
LIN {X 0,Y 449.095,Z 404.212,A -85,B 0,C 180,E1 -8715.093,E2 -8715.093} C_VEL
LIN {X 0,Y 448.489,Z 416.114,A -85,B 0,C 180,E1 -8715.826,E2 -8715.826} C_VEL
LIN {X 0,Y 447.899,Z 427.527,A -85,B 0,C 180,E1 -8716.731,E2 -8716.731} C_VEL
LIN {X 0,Y 447.356,Z 437.853,A -85,B 0,C 180,E1 -8717.755,E2 -8717.755} C_VEL
LIN {X 0,Y 446.759,Z 447.097,A -85,B 0,C 180,E1 -8718.889,E2 -8718.889} C_VEL
LIN {X 0,Y 446.25,Z 456.082,A -85,B 0,C 180,E1 -8720.252,E2 -8720.252} C_VEL
LIN {X 0,Y 445.885,Z 463.316,A -85,B 0,C 180,E1 -8721.616,E2 -8721.616} C_VEL
LIN {X 0,Y 445.674,Z 468.197,A -85,B 0,C 180,E1 -8722.752,E2 -8722.752} C_VEL
LIN {X 0,Y 445.512,Z 472.314,A -85,B 0,C 180,E1 -8723.915,E2 -8723.915} C_VEL
LIN {X 0,Y 445.417,Z 476.565,A -85,B 0,C 180,E1 -8725.474,E2 -8725.474} C_VEL
LIN {X 0,Y 445.357,Z 478.436,A -85,B 0,C 180,E1 -8726.38,E2 -8726.38} C_VEL
LIN {X 0,Y 445.401,Z 479.843,A -85,B 0,C 180,E1 -8727.286,E2 -8727.286} C_VEL
LIN {X 0,Y 445.318,Z 481.454,A -85,B 0,C 180,E1 -8729.095,E2 -8729.095} C_VEL
LIN {X 0,Y 445.319,Z 481.678,A -85,B 0,C 180,E1 -8729.999,E2 -8729.999} C_VEL
LIN {X 0,Y 445.318,Z 481.468,A -85,B 0,C 180,E1 -8730.904,E2 -8730.904} C_VEL
LIN {X 0,Y 445.4,Z 479.874,A -85,B 0,C 180,E1 -8732.712,E2 -8732.712} C_VEL
LIN {X 0,Y 445.357,Z 478.482,A -85,B 0,C 180,E1 -8733.618,E2 -8733.618} C_VEL
LIN {X 0,Y 445.49,Z 475.555,A -85,B 0,C 180,E1 -8734.977,E2 -8734.977} C_VEL
LIN {X 0,Y 445.61,Z 470.162,A -85,B 0,C 180,E1 -8736.747,E2 -8736.747} C_VEL
LIN {X 0,Y 445.855,Z 464.479,A -85,B 0,C 180,E1 -8738.155,E2 -8738.155} C_VEL
LIN {X 0,Y 446.209,Z 457.589,A -85,B 0,C 180,E1 -8739.518,E2 -8739.518} C_VEL
LIN {X 0,Y 446.566,Z 450.556,A -85,B 0,C 180,E1 -8740.656,E2 -8740.656} C_VEL
LIN {X 0,Y 447.144,Z 442.084,A -85,B 0,C 180,E1 -8741.789,E2 -8741.789} C_VEL
LIN {X 0,Y 447.782,Z 432.508,A -85,B 0,C 180,E1 -8742.835,E2 -8742.835} C_VEL
LIN {X 0,Y 448.161,Z 422.686,A -85,B 0,C 180,E1 -8743.72,E2 -8743.72} C_VEL
LIN {X 0,Y 448.768,Z 411.68,A -85,B 0,C 180,E1 -8744.51,E2 -8744.51} C_VEL
LIN {X 0,Y 449.32,Z 399.494,A -85,B 0,C 180,E1 -8745.187,E2 -8745.187} C_VEL
LIN {X 0,Y 449.855,Z 386.759,A -85,B 0,C 180,E1 -8745.691,E2 -8745.691} C_VEL
LIN {X 0,Y 450.173,Z 373.349,A -85,B 0,C 180,E1 -8746.029,E2 -8746.029} C_VEL
LIN {X 0,Y 450.85,Z 289.406,A -85,B 0,C 180,E1 -8747.396,E2 -8747.396} C_VEL
LIN {X 0,Y 447.588,Z 269.863,A -85,B 0,C 180,E1 -8747.876,E2 -8747.876} C_VEL
LIN {X 0,Y 447.697,Z 266.076,A -85,B 0,C 180,E1 -8748.534,E2 -8748.534} C_VEL
LIN {X 0,Y 448.532,Z 248.95,A -85,B 0,C 180,E1 -8751.846,E2 -8751.846} C_VEL
LIN {X 0,Y 448.695,Z 242.833,A -85,B 0,C 180,E1 -8753.052,E2 -8753.052} C_VEL
LIN {X 0,Y 446.49,Z 231.447,A -85,B 0,C 180,E1 -8755.523,E2 -8755.523} C_VEL
LIN {X 0,Y 446.491,Z 231.369,A -85,B 0,C 180,E1 -8758.177,E2 -8758.177} C_VEL
LIN {X 0,Y 446.423,Z 231.377,A -85,B 0,C 180,E1 -8761.773,E2 -8761.773} C_VEL
LIN {X 0,Y 446.432,Z 231.375,A -85,B 0,C 180,E1 -8764.521,E2 -8764.521} C_VEL
LIN {X 0,Y 446.413,Z 231.38,A -85,B 0,C 180,E1 -8768.076,E2 -8768.076} C_VEL
LIN {X 0,Y 446.413,Z 231.373,A -85,B 0,C 180,E1 -8771.391,E2 -8771.391} C_VEL
LIN {X 0,Y 446.424,Z 231.373,A -85,B 0,C 180,E1 -8774.89,E2 -8774.89} C_VEL
LIN {X 0,Y 446.422,Z 231.375,A -85,B 0,C 180,E1 -8777.723,E2 -8777.723} C_VEL
LIN {X 0,Y 446.409,Z 231.373,A -85,B 0,C 180,E1 -8780.967,E2 -8780.967} C_VEL
LIN {X 0,Y 446.416,Z 231.378,A -85,B 0,C 180,E1 -8784.371,E2 -8784.371} C_VEL
LIN {X 0,Y 446.417,Z 231.372,A -85,B 0,C 180,E1 -8787.636,E2 -8787.636} C_VEL
LIN {X 0,Y 446.421,Z 231.379,A -85,B 0,C 180,E1 -8790.786,E2 -8790.786} C_VEL
LIN {X 0,Y 446.434,Z 231.37,A -85,B 0,C 180,E1 -8793.843,E2 -8793.843} C_VEL
LIN {X 0,Y 446.421,Z 231.374,A -85,B 0,C 180,E1 -8796.82,E2 -8796.82} C_VEL
LIN {X 0,Y 446.44,Z 231.371,A -85,B 0,C 180,E1 -8799.734,E2 -8799.734} C_VEL
LIN {X 0,Y 446.449,Z 231.366,A -85,B 0,C 180,E1 -8802.594,E2 -8802.594} C_VEL
LIN {X 0,Y 446.456,Z 231.369,A -85,B 0,C 180,E1 -8805.409,E2 -8805.409} C_VEL
LIN {X 0,Y 446.51,Z 231.361,A -85,B 0,C 180,E1 -8808.19,E2 -8808.19} C_VEL
LIN {X 0,Y 446.505,Z 231.364,A -85,B 0,C 180,E1 -8810.941,E2 -8810.941} C_VEL
LIN {X 0,Y 446.616,Z 231.353,A -85,B 0,C 180,E1 -8813.673,E2 -8813.673} C_VEL
LIN {X 0,Y 446.64,Z 231.345,A -85,B 0,C 180,E1 -8817.291,E2 -8817.291} C_VEL
LIN {X 0,Y 446.667,Z 231.341,A -85,B 0,C 180,E1 -8819.997,E2 -8819.997} C_VEL
LIN {X 0,Y 446.626,Z 231.347,A -85,B 0,C 180,E1 -8822.703,E2 -8822.703} C_VEL
LIN {X 0,Y 446.585,Z 231.353,A -85,B 0,C 180,E1 -8826.321,E2 -8826.321} C_VEL
LIN {X 0,Y 446.495,Z 231.363,A -85,B 0,C 180,E1 -8829.053,E2 -8829.053} C_VEL
LIN {X 0,Y 446.507,Z 231.361,A -85,B 0,C 180,E1 -8832.727,E2 -8832.727} C_VEL
LIN {X 0,Y 446.471,Z 231.367,A -85,B 0,C 180,E1 -8836.456,E2 -8836.456} C_VEL
LIN {X 0,Y 446.45,Z 231.37,A -85,B 0,C 180,E1 -8839.3,E2 -8839.3} C_VEL
LIN {X 0,Y 446.399,Z 231.381,A -85,B 0,C 180,E1 -8842.196,E2 -8842.196} C_VEL
LIN {X 0,Y 446.421,Z 231.372,A -85,B 0,C 180,E1 -8845.15,E2 -8845.15} C_VEL
LIN {X 0,Y 446.426,Z 231.373,A -85,B 0,C 180,E1 -8848.178,E2 -8848.178} C_VEL
LIN {X 0,Y 446.39,Z 231.377,A -85,B 0,C 180,E1 -8851.298,E2 -8851.298} C_VEL
LIN {X 0,Y 446.405,Z 231.379,A -85,B 0,C 180,E1 -8854.52,E2 -8854.52} C_VEL
LIN {X 0,Y 446.41,Z 231.377,A -85,B 0,C 180,E1 -8858.08,E2 -8858.08} C_VEL
LIN {X 0,Y 446.419,Z 231.378,A -85,B 0,C 180,E1 -8860.918,E2 -8860.918} C_VEL
LIN {X 0,Y 446.475,Z 231.513,A -85,B 0,C 180,E1 -8863.716,E2 -8863.716} C_VEL
LIN {X 0,Y 448.077,Z 239.724,A -85,B 0,C 180,E1 -8865.526,E2 -8865.526} C_VEL
LIN {X 0,Y 448.065,Z 246.916,A -85,B 0,C 180,E1 -8866.978,E2 -8866.978} C_VEL
LIN {X 0,Y 447.6,Z 258.034,A -85,B 0,C 180,E1 -8869.138,E2 -8869.138} C_VEL
LIN {X 0,Y 448.449,Z 262.515,A -85,B 0,C 180,E1 -8869.292,E2 -8869.292} C_VEL
LIN {X 0,Y 451.048,Z 277.085,A -85,B 0,C 180,E1 -8869.647,E2 -8869.647} C_VEL
LIN {X 0,Y 450.092,Z 365.656,A -85,B 0,C 180,E1 -8871.099,E2 -8871.099} C_VEL
LIN {X 0,Y 449.745,Z 379.15,A -85,B 0,C 180,E1 -8871.506,E2 -8871.506} C_VEL
LIN {X 0,Y 449.341,Z 391.466,A -85,B 0,C 180,E1 -8872.059,E2 -8872.059} C_VEL
LIN {X 0,Y 448.824,Z 402.916,A -85,B 0,C 180,E1 -8872.749,E2 -8872.749} C_VEL
LIN {X 0,Y 448.122,Z 415.035,A -85,B 0,C 180,E1 -8873.699,E2 -8873.699} C_VEL
LIN {X 0,Y 447.509,Z 425.582,A -85,B 0,C 180,E1 -8874.742,E2 -8874.742} C_VEL
LIN {X 0,Y 447.02,Z 434.228,A -85,B 0,C 180,E1 -8875.796,E2 -8875.796} C_VEL
LIN {X 0,Y 446.479,Z 442.99,A -85,B 0,C 180,E1 -8877.109,E2 -8877.109} C_VEL
LIN {X 0,Y 446.118,Z 449.394,A -85,B 0,C 180,E1 -8878.279,E2 -8878.279} C_VEL
LIN {X 0,Y 445.841,Z 455.726,A -85,B 0,C 180,E1 -8879.708,E2 -8879.708} C_VEL
LIN {X 0,Y 445.565,Z 461.038,A -85,B 0,C 180,E1 -8881.245,E2 -8881.245} C_VEL
LIN {X 0,Y 445.417,Z 464.908,A -85,B 0,C 180,E1 -8882.77,E2 -8882.77} C_VEL
LIN {X 0,Y 445.275,Z 467.271,A -85,B 0,C 180,E1 -8884.102,E2 -8884.102} C_VEL
LIN {X 0,Y 445.182,Z 468.944,A -85,B 0,C 180,E1 -8885.768,E2 -8885.768} C_VEL
LIN {X 0,Y 445.175,Z 469.242,A -85,B 0,C 180,E1 -8886.44,E2 -8886.44} C_VEL
LIN {X 0,Y 444.498,Z 469.33,A -85,B 0,C 180,E1 -8887.196,E2 -8887.196} C_VEL
LIN {X 0,Y 441.639,Z 468.94,A -85,B 0,C 180,E1 -8888.424,E2 -8888.424} C_VEL
LIN {X 0,Y 439.257,Z 468.111,A -85,B 0,C 180,E1 -8889.408,E2 -8889.408} C_VEL
LIN {X 0,Y 438.271,Z 467.096,A -85,B 0,C 180,E1 -8890.161,E2 -8890.161} C_VEL
LIN {X 0,Y 438.211,Z 466.674,A -85,B 0,C 180,E1 -8890.414,E2 -8890.414} C_VEL
LIN {X 0,Y 438.368,Z 463.999,A -85,B 0,C 180,E1 -8891.783,E2 -8891.783} C_VEL
LIN {X 0,Y 438.506,Z 460.064,A -85,B 0,C 180,E1 -8893.233,E2 -8893.233} C_VEL
LIN {X 0,Y 438.813,Z 454.917,A -85,B 0,C 180,E1 -8894.678,E2 -8894.678} C_VEL
LIN {X 0,Y 439.113,Z 448.452,A -85,B 0,C 180,E1 -8896.11,E2 -8896.11} C_VEL
LIN {X 0,Y 439.566,Z 441.279,A -85,B 0,C 180,E1 -8897.385,E2 -8897.385} C_VEL
LIN {X 0,Y 440.127,Z 431.979,A -85,B 0,C 180,E1 -8898.721,E2 -8898.721} C_VEL
LIN {X 0,Y 440.738,Z 421.825,A -85,B 0,C 180,E1 -8899.899,E2 -8899.899} C_VEL
LIN {X 0,Y 441.367,Z 411.729,A -85,B 0,C 180,E1 -8900.838,E2 -8900.838} C_VEL
LIN {X 0,Y 441.966,Z 400.667,A -85,B 0,C 180,E1 -8901.661,E2 -8901.661} C_VEL
LIN {X 0,Y 442.467,Z 388.638,A -85,B 0,C 180,E1 -8902.356,E2 -8902.356} C_VEL
LIN {X 0,Y 442.861,Z 376.304,A -85,B 0,C 180,E1 -8902.879,E2 -8902.879} C_VEL
LIN {X 0,Y 443.237,Z 363.424,A -85,B 0,C 180,E1 -8903.228,E2 -8903.228} C_VEL
LIN {X 0,Y 444.004,Z 276.637,A -85,B 0,C 180,E1 -8904.665,E2 -8904.665} C_VEL
LIN {X 0,Y 440.742,Z 258.831,A -85,B 0,C 180,E1 -8905.113,E2 -8905.113} C_VEL
LIN {X 0,Y 440.699,Z 258.038,A -85,B 0,C 180,E1 -8905.198,E2 -8905.198} C_VEL
LIN {X 0,Y 441.379,Z 244.055,A -85,B 0,C 180,E1 -8908.176,E2 -8908.176} C_VEL
LIN {X 0,Y 440.359,Z 236.01,A -85,B 0,C 180,E1 -8910.001,E2 -8910.001} C_VEL
LIN {X 0,Y 439.636,Z 232.277,A -85,B 0,C 180,E1 -8910.917,E2 -8910.917} C_VEL
LIN {X 0,Y 439.62,Z 232.224,A -85,B 0,C 180,E1 -8912.75,E2 -8912.75} C_VEL
LIN {X 0,Y 439.58,Z 232.225,A -85,B 0,C 180,E1 -8916.426,E2 -8916.426} C_VEL
LIN {X 0,Y 439.463,Z 232.242,A -85,B 0,C 180,E1 -8919.203,E2 -8919.203} C_VEL
LIN {X 0,Y 439.468,Z 232.233,A -85,B 0,C 180,E1 -8922.728,E2 -8922.728} C_VEL
LIN {X 0,Y 439.412,Z 232.246,A -85,B 0,C 180,E1 -8926.35,E2 -8926.35} C_VEL
LIN {X 0,Y 439.368,Z 232.255,A -85,B 0,C 180,E1 -8929.628,E2 -8929.628} C_VEL
LIN {X 0,Y 439.33,Z 232.257,A -85,B 0,C 180,E1 -8932.578,E2 -8932.578} C_VEL
LIN {X 0,Y 439.347,Z 232.254,A -85,B 0,C 180,E1 -8935.589,E2 -8935.589} C_VEL
LIN {X 0,Y 439.368,Z 232.246,A -85,B 0,C 180,E1 -8938.678,E2 -8938.678} C_VEL
LIN {X 0,Y 439.336,Z 232.259,A -85,B 0,C 180,E1 -8942.032,E2 -8942.032} C_VEL
LIN {X 0,Y 439.36,Z 232.243,A -85,B 0,C 180,E1 -8945.342,E2 -8945.342} C_VEL
LIN {X 0,Y 439.33,Z 232.263,A -85,B 0,C 180,E1 -8948.601,E2 -8948.601} C_VEL
LIN {X 0,Y 439.326,Z 232.252,A -85,B 0,C 180,E1 -8952.213,E2 -8952.213} C_VEL
LIN {X 0,Y 439.374,Z 232.252,A -85,B 0,C 180,E1 -8955.274,E2 -8955.274} C_VEL
LIN {X 0,Y 439.332,Z 232.254,A -85,B 0,C 180,E1 -8959.02,E2 -8959.02} C_VEL
LIN {X 0,Y 439.327,Z 232.247,A -85,B 0,C 180,E1 -8962.568,E2 -8962.568} C_VEL
LIN {X 0,Y 439.379,Z 232.252,A -85,B 0,C 180,E1 -8964.847,E2 -8964.847} C_VEL
LIN {X 0,Y 439.35,Z 232.25,A -85,B 0,C 180,E1 -8968.143,E2 -8968.143} C_VEL
LIN {X 0,Y 439.373,Z 232.239,A -85,B 0,C 180,E1 -8971.613,E2 -8971.613} C_VEL
LIN {X 0,Y 439.35,Z 232.249,A -85,B 0,C 180,E1 -8974.416,E2 -8974.416} C_VEL
LIN {X 0,Y 439.353,Z 232.26,A -85,B 0,C 180,E1 -8977.428,E2 -8977.428} C_VEL
LIN {X 0,Y 439.433,Z 232.233,A -85,B 0,C 180,E1 -8980.667,E2 -8980.667} C_VEL
LIN {X 0,Y 439.455,Z 232.233,A -85,B 0,C 180,E1 -8984.228,E2 -8984.228} C_VEL
LIN {X 0,Y 439.472,Z 232.243,A -85,B 0,C 180,E1 -8988.005,E2 -8988.005} C_VEL
LIN {X 0,Y 439.481,Z 232.235,A -85,B 0,C 180,E1 -8991.728,E2 -8991.728} C_VEL
LIN {X 0,Y 439.596,Z 232.209,A -85,B 0,C 180,E1 -8994.499,E2 -8994.499} C_VEL
LIN {X 0,Y 439.629,Z 232.223,A -85,B 0,C 180,E1 -8998.171,E2 -8998.171} C_VEL
LIN {X 0,Y 439.577,Z 232.223,A -85,B 0,C 180,E1 -9000.919,E2 -9000.919} C_VEL
LIN {X 0,Y 439.605,Z 232.215,A -85,B 0,C 180,E1 -9002.752,E2 -9002.752} C_VEL
LIN {X 0,Y 439.597,Z 232.214,A -85,B 0,C 180,E1 -9006.428,E2 -9006.428} C_VEL
LIN {X 0,Y 439.49,Z 232.236,A -85,B 0,C 180,E1 -9009.205,E2 -9009.205} C_VEL
LIN {X 0,Y 439.472,Z 232.235,A -85,B 0,C 180,E1 -9012.94,E2 -9012.94} C_VEL
LIN {X 0,Y 439.454,Z 232.23,A -85,B 0,C 180,E1 -9016.35,E2 -9016.35} C_VEL
LIN {X 0,Y 439.41,Z 232.246,A -85,B 0,C 180,E1 -9019.628,E2 -9019.628} C_VEL
LIN {X 0,Y 439.371,Z 232.252,A -85,B 0,C 180,E1 -9022.578,E2 -9022.578} C_VEL
LIN {X 0,Y 439.385,Z 232.247,A -85,B 0,C 180,E1 -9025.589,E2 -9025.589} C_VEL
LIN {X 0,Y 439.4,Z 232.25,A -85,B 0,C 180,E1 -9028.677,E2 -9028.677} C_VEL
LIN {X 0,Y 439.375,Z 232.245,A -85,B 0,C 180,E1 -9032.031,E2 -9032.031} C_VEL
LIN {X 0,Y 439.401,Z 232.253,A -85,B 0,C 180,E1 -9035.341,E2 -9035.341} C_VEL
LIN {X 0,Y 439.372,Z 232.248,A -85,B 0,C 180,E1 -9038.599,E2 -9038.599} C_VEL
LIN {X 0,Y 439.369,Z 232.246,A -85,B 0,C 180,E1 -9042.21,E2 -9042.21} C_VEL
LIN {X 0,Y 439.386,Z 232.253,A -85,B 0,C 180,E1 -9045.268,E2 -9045.268} C_VEL
LIN {X 0,Y 439.377,Z 232.25,A -85,B 0,C 180,E1 -9048.747,E2 -9048.747} C_VEL
LIN {X 0,Y 439.374,Z 232.257,A -85,B 0,C 180,E1 -9051.61,E2 -9051.61} C_VEL
LIN {X 0,Y 439.408,Z 232.248,A -85,B 0,C 180,E1 -9054.844,E2 -9054.844} C_VEL
LIN {X 0,Y 439.383,Z 232.257,A -85,B 0,C 180,E1 -9058.14,E2 -9058.14} C_VEL
LIN {X 0,Y 439.444,Z 232.244,A -85,B 0,C 180,E1 -9061.598,E2 -9061.598} C_VEL
LIN {X 0,Y 439.478,Z 232.423,A -85,B 0,C 180,E1 -9064.238,E2 -9064.238} C_VEL
LIN {X 0,Y 441.658,Z 243.953,A -85,B 0,C 180,E1 -9066.775,E2 -9066.775} C_VEL
LIN {X 0,Y 441.773,Z 247.731,A -85,B 0,C 180,E1 -9067.554,E2 -9067.554} C_VEL
LIN {X 0,Y 440.818,Z 264.615,A -85,B 0,C 180,E1 -9070.923,E2 -9070.923} C_VEL
LIN {X 0,Y 440.581,Z 269.834,A -85,B 0,C 180,E1 -9071.905,E2 -9071.905} C_VEL
LIN {X 0,Y 444.051,Z 291.225,A -85,B 0,C 180,E1 -9072.429,E2 -9072.429} C_VEL
LIN {X 0,Y 443.158,Z 377.397,A -85,B 0,C 180,E1 -9073.857,E2 -9073.857} C_VEL
LIN {X 0,Y 442.711,Z 390.652,A -85,B 0,C 180,E1 -9074.254,E2 -9074.254} C_VEL
LIN {X 0,Y 442.231,Z 403.942,A -85,B 0,C 180,E1 -9074.856,E2 -9074.856} C_VEL
LIN {X 0,Y 441.569,Z 415.888,A -85,B 0,C 180,E1 -9075.6,E2 -9075.6} C_VEL
LIN {X 0,Y 440.989,Z 426.578,A -85,B 0,C 180,E1 -9076.452,E2 -9076.452} C_VEL
LIN {X 0,Y 440.407,Z 437.674,A -85,B 0,C 180,E1 -9077.558,E2 -9077.558} C_VEL
LIN {X 0,Y 439.761,Z 446.939,A -85,B 0,C 180,E1 -9078.709,E2 -9078.709} C_VEL
LIN {X 0,Y 439.235,Z 455.938,A -85,B 0,C 180,E1 -9080.095,E2 -9080.095} C_VEL
LIN {X 0,Y 438.847,Z 463.184,A -85,B 0,C 180,E1 -9081.48,E2 -9081.48} C_VEL
LIN {X 0,Y 438.614,Z 468.073,A -85,B 0,C 180,E1 -9082.635,E2 -9082.635} C_VEL
LIN {X 0,Y 438.413,Z 472.62,A -85,B 0,C 180,E1 -9083.953,E2 -9083.953} C_VEL
LIN {X 0,Y 438.348,Z 476.454,A -85,B 0,C 180,E1 -9085.401,E2 -9085.401} C_VEL
LIN {X 0,Y 438.262,Z 478.328,A -85,B 0,C 180,E1 -9086.322,E2 -9086.322} C_VEL
LIN {X 0,Y 438.296,Z 479.738,A -85,B 0,C 180,E1 -9087.242,E2 -9087.242} C_VEL
LIN {X 0,Y 438.276,Z 480.74,A -85,B 0,C 180,E1 -9088.161,E2 -9088.161} C_VEL
LIN {X 0,Y 438.231,Z 481.579,A -85,B 0,C 180,E1 -9089.999,E2 -9089.999} C_VEL
LIN {X 0,Y 438.233,Z 481.372,A -85,B 0,C 180,E1 -9090.918,E2 -9090.918} C_VEL
LIN {X 0,Y 438.276,Z 480.77,A -85,B 0,C 180,E1 -9091.837,E2 -9091.837} C_VEL
LIN {X 0,Y 438.296,Z 479.78,A -85,B 0,C 180,E1 -9092.756,E2 -9092.756} C_VEL
LIN {X 0,Y 438.262,Z 478.391,A -85,B 0,C 180,E1 -9093.677,E2 -9093.677} C_VEL
LIN {X 0,Y 438.422,Z 475.467,A -85,B 0,C 180,E1 -9095.057,E2 -9095.057} C_VEL
LIN {X 0,Y 438.472,Z 471.505,A -85,B 0,C 180,E1 -9096.441,E2 -9096.441} C_VEL
LIN {X 0,Y 438.747,Z 465.416,A -85,B 0,C 180,E1 -9098.056,E2 -9098.056} C_VEL
LIN {X 0,Y 439.101,Z 458.757,A -85,B 0,C 180,E1 -9099.442,E2 -9099.442} C_VEL
LIN {X 0,Y 439.561,Z 450.492,A -85,B 0,C 180,E1 -9100.827,E2 -9100.827} C_VEL
LIN {X 0,Y 440.176,Z 442.028,A -85,B 0,C 180,E1 -9101.979,E2 -9101.979} C_VEL
LIN {X 0,Y 440.872,Z 431.389,A -85,B 0,C 180,E1 -9103.147,E2 -9103.147} C_VEL
LIN {X 0,Y 441.362,Z 421.226,A -85,B 0,C 180,E1 -9104.053,E2 -9104.053} C_VEL
LIN {X 0,Y 442.009,Z 409.896,A -85,B 0,C 180,E1 -9104.855,E2 -9104.855} C_VEL
LIN {X 0,Y 442.555,Z 398.317,A -85,B 0,C 180,E1 -9105.484,E2 -9105.484} C_VEL
LIN {X 0,Y 443.091,Z 385.011,A -85,B 0,C 180,E1 -9105.996,E2 -9105.996} C_VEL
LIN {X 0,Y 443.416,Z 372.052,A -85,B 0,C 180,E1 -9106.309,E2 -9106.309} C_VEL
LIN {X 0,Y 444.072,Z 289.912,A -85,B 0,C 180,E1 -9107.668,E2 -9107.668} C_VEL
LIN {X 0,Y 440.626,Z 269.517,A -85,B 0,C 180,E1 -9108.196,E2 -9108.196} C_VEL
LIN {X 0,Y 441.463,Z 252.56,A -85,B 0,C 180,E1 -9111.478,E2 -9111.478} C_VEL
LIN {X 0,Y 441.8,Z 244.959,A -85,B 0,C 180,E1 -9112.989,E2 -9112.989} C_VEL
LIN {X 0,Y 439.573,Z 232.954,A -85,B 0,C 180,E1 -9115.573,E2 -9115.573} C_VEL
LIN {X 0,Y 439.443,Z 232.27,A -85,B 0,C 180,E1 -9115.823,E2 -9115.823} C_VEL
LIN {X 0,Y 439.422,Z 232.249,A -85,B 0,C 180,E1 -9118.672,E2 -9118.672} C_VEL
LIN {X 0,Y 439.374,Z 232.256,A -85,B 0,C 180,E1 -9122.028,E2 -9122.028} C_VEL
LIN {X 0,Y 439.397,Z 232.251,A -85,B 0,C 180,E1 -9125.338,E2 -9125.338} C_VEL
LIN {X 0,Y 439.365,Z 232.254,A -85,B 0,C 180,E1 -9128.595,E2 -9128.595} C_VEL
LIN {X 0,Y 439.385,Z 232.257,A -85,B 0,C 180,E1 -9132.204,E2 -9132.204} C_VEL
LIN {X 0,Y 439.379,Z 232.25,A -85,B 0,C 180,E1 -9135.265,E2 -9135.265} C_VEL
LIN {X 0,Y 439.372,Z 232.255,A -85,B 0,C 180,E1 -9138.744,E2 -9138.744} C_VEL
LIN {X 0,Y 439.365,Z 232.249,A -85,B 0,C 180,E1 -9141.607,E2 -9141.607} C_VEL
LIN {X 0,Y 439.395,Z 232.25,A -85,B 0,C 180,E1 -9144.841,E2 -9144.841} C_VEL
LIN {X 0,Y 439.369,Z 232.253,A -85,B 0,C 180,E1 -9148.137,E2 -9148.137} C_VEL
LIN {X 0,Y 439.399,Z 232.246,A -85,B 0,C 180,E1 -9151.604,E2 -9151.604} C_VEL
LIN {X 0,Y 439.365,Z 232.253,A -85,B 0,C 180,E1 -9154.41,E2 -9154.41} C_VEL
LIN {X 0,Y 439.36,Z 232.252,A -85,B 0,C 180,E1 -9157.422,E2 -9157.422} C_VEL
LIN {X 0,Y 439.438,Z 232.246,A -85,B 0,C 180,E1 -9160.661,E2 -9160.661} C_VEL
LIN {X 0,Y 439.456,Z 232.241,A -85,B 0,C 180,E1 -9164.222,E2 -9164.222} C_VEL
LIN {X 0,Y 439.477,Z 232.237,A -85,B 0,C 180,E1 -9167.998,E2 -9167.998} C_VEL
LIN {X 0,Y 439.474,Z 232.238,A -85,B 0,C 180,E1 -9171.722,E2 -9171.722} C_VEL
LIN {X 0,Y 439.599,Z 232.223,A -85,B 0,C 180,E1 -9174.493,E2 -9174.493} C_VEL
LIN {X 0,Y 439.614,Z 232.222,A -85,B 0,C 180,E1 -9178.165,E2 -9178.165} C_VEL
LIN {X 0,Y 439.619,Z 232.219,A -85,B 0,C 180,E1 -9179.997,E2 -9179.997} C_VEL
LIN {X 0,Y 439.58,Z 232.224,A -85,B 0,C 180,E1 -9182.746,E2 -9182.746} C_VEL
LIN {X 0,Y 439.537,Z 232.23,A -85,B 0,C 180,E1 -9186.423,E2 -9186.423} C_VEL
LIN {X 0,Y 439.461,Z 232.24,A -85,B 0,C 180,E1 -9189.199,E2 -9189.199} C_VEL
LIN {X 0,Y 439.45,Z 232.24,A -85,B 0,C 180,E1 -9192.934,E2 -9192.934} C_VEL
LIN {X 0,Y 439.429,Z 232.245,A -85,B 0,C 180,E1 -9196.344,E2 -9196.344} C_VEL
LIN {X 0,Y 439.383,Z 232.253,A -85,B 0,C 180,E1 -9199.623,E2 -9199.623} C_VEL
LIN {X 0,Y 439.344,Z 232.256,A -85,B 0,C 180,E1 -9202.572,E2 -9202.572} C_VEL
LIN {X 0,Y 439.358,Z 232.252,A -85,B 0,C 180,E1 -9205.583,E2 -9205.583} C_VEL
LIN {X 0,Y 439.377,Z 232.249,A -85,B 0,C 180,E1 -9208.672,E2 -9208.672} C_VEL
LIN {X 0,Y 439.345,Z 232.256,A -85,B 0,C 180,E1 -9212.027,E2 -9212.027} C_VEL
LIN {X 0,Y 439.37,Z 232.253,A -85,B 0,C 180,E1 -9215.338,E2 -9215.338} C_VEL
LIN {X 0,Y 439.37,Z 232.258,A -85,B 0,C 180,E1 -9218.591,E2 -9218.591} C_VEL
LIN {X 0,Y 439.376,Z 232.257,A -85,B 0,C 180,E1 -9221.257,E2 -9221.257} C_VEL
LIN {X 0,Y 439.403,Z 232.328,A -85,B 0,C 180,E1 -9223.447,E2 -9223.447} C_VEL
LIN {X 0,Y 440.417,Z 237.234,A -85,B 0,C 180,E1 -9224.592,E2 -9224.592} C_VEL
LIN {X 0,Y 441.302,Z 242.714,A -85,B 0,C 180,E1 -9225.772,E2 -9225.772} C_VEL
LIN {X 0,Y 440.694,Z 257.822,A -85,B 0,C 180,E1 -9228.8,E2 -9228.8} C_VEL
LIN {X 0,Y 440.871,Z 259.353,A -85,B 0,C 180,E1 -9228.903,E2 -9228.903} C_VEL
LIN {X 0,Y 444.234,Z 277.378,A -85,B 0,C 180,E1 -9229.367,E2 -9229.367} C_VEL
LIN {X 0,Y 443.276,Z 365.992,A -85,B 0,C 180,E1 -9230.847,E2 -9230.847} C_VEL
LIN {X 0,Y 442.919,Z 379.34,A -85,B 0,C 180,E1 -9231.258,E2 -9231.258} C_VEL
LIN {X 0,Y 442.515,Z 391.242,A -85,B 0,C 180,E1 -9231.799,E2 -9231.799} C_VEL
LIN {X 0,Y 441.96,Z 402.919,A -85,B 0,C 180,E1 -9232.509,E2 -9232.509} C_VEL
LIN {X 0,Y 441.239,Z 414.976,A -85,B 0,C 180,E1 -9233.467,E2 -9233.467} C_VEL
LIN {X 0,Y 440.555,Z 425.971,A -85,B 0,C 180,E1 -9234.572,E2 -9234.572} C_VEL
LIN {X 0,Y 439.991,Z 435.207,A -85,B 0,C 180,E1 -9235.734,E2 -9235.734} C_VEL
LIN {X 0,Y 439.443,Z 443.781,A -85,B 0,C 180,E1 -9237.061,E2 -9237.061} C_VEL
LIN {X 0,Y 439.004,Z 450.699,A -85,B 0,C 180,E1 -9238.38,E2 -9238.38} C_VEL
LIN {X 0,Y 438.725,Z 456.962,A -85,B 0,C 180,E1 -9239.877,E2 -9239.877} C_VEL
LIN {X 0,Y 438.491,Z 461.475,A -85,B 0,C 180,E1 -9241.261,E2 -9241.261} C_VEL
LIN {X 0,Y 438.323,Z 465.229,A -85,B 0,C 180,E1 -9242.81,E2 -9242.81} C_VEL
LIN {X 0,Y 438.15,Z 467.733,A -85,B 0,C 180,E1 -9244.338,E2 -9244.338} C_VEL
LIN {X 0,Y 438.09,Z 469.233,A -85,B 0,C 180,E1 -9246.11,E2 -9246.11} C_VEL
LIN {X 0,Y 438.075,Z 469.39,A -85,B 0,C 180,E1 -9247.355,E2 -9247.355} C_VEL
LIN {X 0,Y 438.098,Z 468.932,A -85,B 0,C 180,E1 -9248.49,E2 -9248.49} C_VEL
LIN {X 0,Y 438.122,Z 468.169,A -85,B 0,C 180,E1 -9249.336,E2 -9249.336} C_VEL
LIN {X 0,Y 438.211,Z 466.674,A -85,B 0,C 180,E1 -9250.414,E2 -9250.414} C_VEL
LIN {X 0,Y 437.606,Z 465.379,A -85,B 0,C 180,E1 -9251.161,E2 -9251.161} C_VEL
LIN {X 0,Y 434.837,Z 462.722,A -85,B 0,C 180,E1 -9252.364,E2 -9252.364} C_VEL
LIN {X 0,Y 432.531,Z 460.139,A -85,B 0,C 180,E1 -9253.315,E2 -9253.315} C_VEL
LIN {X 0,Y 431.63,Z 457.843,A -85,B 0,C 180,E1 -9254.032,E2 -9254.032} C_VEL
LIN {X 0,Y 431.606,Z 456.991,A -85,B 0,C 180,E1 -9254.271,E2 -9254.271} C_VEL
LIN {X 0,Y 431.94,Z 451.475,A -85,B 0,C 180,E1 -9255.634,E2 -9255.634} C_VEL
LIN {X 0,Y 432.302,Z 445.43,A -85,B 0,C 180,E1 -9256.845,E2 -9256.845} C_VEL
LIN {X 0,Y 432.752,Z 438.166,A -85,B 0,C 180,E1 -9258.051,E2 -9258.051} C_VEL
LIN {X 0,Y 433.32,Z 429.345,A -85,B 0,C 180,E1 -9259.251,E2 -9259.251} C_VEL
LIN {X 0,Y 434.026,Z 418.446,A -85,B 0,C 180,E1 -9260.447,E2 -9260.447} C_VEL
LIN {X 0,Y 434.722,Z 407.053,A -85,B 0,C 180,E1 -9261.439,E2 -9261.439} C_VEL
LIN {X 0,Y 435.355,Z 394.365,A -85,B 0,C 180,E1 -9262.289,E2 -9262.289} C_VEL
LIN {X 0,Y 435.814,Z 382.64,A -85,B 0,C 180,E1 -9262.88,E2 -9262.88} C_VEL
LIN {X 0,Y 436.25,Z 370.042,A -85,B 0,C 180,E1 -9263.323,E2 -9263.323} C_VEL
LIN {X 0,Y 436.529,Z 354.104,A -85,B 0,C 180,E1 -9263.646,E2 -9263.646} C_VEL
LIN {X 0,Y 437.251,Z 277.593,A -85,B 0,C 180,E1 -9264.924,E2 -9264.924} C_VEL
LIN {X 0,Y 433.776,Z 258.774,A -85,B 0,C 180,E1 -9265.412,E2 -9265.412} C_VEL
LIN {X 0,Y 433.791,Z 256.538,A -85,B 0,C 180,E1 -9265.82,E2 -9265.82} C_VEL
LIN {X 0,Y 434.431,Z 244.776,A -85,B 0,C 180,E1 -9268.378,E2 -9268.378} C_VEL
LIN {X 0,Y 433.142,Z 235.77,A -85,B 0,C 180,E1 -9270.466,E2 -9270.466} C_VEL
LIN {X 0,Y 432.563,Z 233.128,A -85,B 0,C 180,E1 -9271.164,E2 -9271.164} C_VEL
LIN {X 0,Y 432.57,Z 233.102,A -85,B 0,C 180,E1 -9272.795,E2 -9272.795} C_VEL
LIN {X 0,Y 432.535,Z 233.103,A -85,B 0,C 180,E1 -9276.532,E2 -9276.532} C_VEL
LIN {X 0,Y 432.407,Z 233.12,A -85,B 0,C 180,E1 -9279.355,E2 -9279.355} C_VEL
LIN {X 0,Y 432.409,Z 233.112,A -85,B 0,C 180,E1 -9282.813,E2 -9282.813} C_VEL
LIN {X 0,Y 432.378,Z 233.121,A -85,B 0,C 180,E1 -9286.481,E2 -9286.481} C_VEL
LIN {X 0,Y 432.304,Z 233.134,A -85,B 0,C 180,E1 -9289.963,E2 -9289.963} C_VEL
LIN {X 0,Y 432.284,Z 233.133,A -85,B 0,C 180,E1 -9292.967,E2 -9292.967} C_VEL
LIN {X 0,Y 432.307,Z 233.129,A -85,B 0,C 180,E1 -9295.005,E2 -9295.005} C_VEL
LIN {X 0,Y 432.316,Z 233.132,A -85,B 0,C 180,E1 -9298.129,E2 -9298.129} C_VEL
LIN {X 0,Y 432.289,Z 233.133,A -85,B 0,C 180,E1 -9301.349,E2 -9301.349} C_VEL
LIN {X 0,Y 432.298,Z 233.127,A -85,B 0,C 180,E1 -9304.682,E2 -9304.682} C_VEL
LIN {X 0,Y 432.297,Z 233.135,A -85,B 0,C 180,E1 -9308.155,E2 -9308.155} C_VEL
LIN {X 0,Y 432.279,Z 233.127,A -85,B 0,C 180,E1 -9311.804,E2 -9311.804} C_VEL
LIN {X 0,Y 432.31,Z 233.126,A -85,B 0,C 180,E1 -9314.351,E2 -9314.351} C_VEL
LIN {X 0,Y 432.28,Z 233.138,A -85,B 0,C 180,E1 -9317.022,E2 -9317.022} C_VEL
LIN {X 0,Y 432.269,Z 233.127,A -85,B 0,C 180,E1 -9319.832,E2 -9319.832} C_VEL
LIN {X 0,Y 432.287,Z 233.129,A -85,B 0,C 180,E1 -9323.026,E2 -9323.026} C_VEL
LIN {X 0,Y 432.317,Z 233.129,A -85,B 0,C 180,E1 -9326.006,E2 -9326.006} C_VEL
LIN {X 0,Y 432.326,Z 233.12,A -85,B 0,C 180,E1 -9329.495,E2 -9329.495} C_VEL
LIN {X 0,Y 432.305,Z 233.118,A -85,B 0,C 180,E1 -9331.876,E2 -9331.876} C_VEL
LIN {X 0,Y 432.308,Z 233.129,A -85,B 0,C 180,E1 -9335.001,E2 -9335.001} C_VEL
LIN {X 0,Y 432.348,Z 233.125,A -85,B 0,C 180,E1 -9338.049,E2 -9338.049} C_VEL
LIN {X 0,Y 432.376,Z 233.114,A -85,B 0,C 180,E1 -9341.033,E2 -9341.033} C_VEL
LIN {X 0,Y 432.423,Z 233.109,A -85,B 0,C 180,E1 -9343.965,E2 -9343.965} C_VEL
LIN {X 0,Y 432.45,Z 233.12,A -85,B 0,C 180,E1 -9347.807,E2 -9347.807} C_VEL
LIN {X 0,Y 432.447,Z 233.112,A -85,B 0,C 180,E1 -9351.593,E2 -9351.593} C_VEL
LIN {X 0,Y 432.551,Z 233.086,A -85,B 0,C 180,E1 -9354.409,E2 -9354.409} C_VEL
LIN {X 0,Y 432.598,Z 233.098,A -85,B 0,C 180,E1 -9358.141,E2 -9358.141} C_VEL
LIN {X 0,Y 432.539,Z 233.1,A -85,B 0,C 180,E1 -9360.934,E2 -9360.934} C_VEL
LIN {X 0,Y 432.559,Z 233.092,A -85,B 0,C 180,E1 -9362.797,E2 -9362.797} C_VEL
LIN {X 0,Y 432.583,Z 233.078,A -85,B 0,C 180,E1 -9365.597,E2 -9365.597} C_VEL
LIN {X 0,Y 432.466,Z 233.112,A -85,B 0,C 180,E1 -9368.413,E2 -9368.413} C_VEL
LIN {X 0,Y 432.465,Z 233.113,A -85,B 0,C 180,E1 -9372.199,E2 -9372.199} C_VEL
LIN {X 0,Y 432.437,Z 233.101,A -85,B 0,C 180,E1 -9376.041,E2 -9376.041} C_VEL
LIN {X 0,Y 432.395,Z 233.121,A -85,B 0,C 180,E1 -9379.487,E2 -9379.487} C_VEL
LIN {X 0,Y 432.324,Z 233.123,A -85,B 0,C 180,E1 -9382.967,E2 -9382.967} C_VEL
LIN {X 0,Y 432.346,Z 233.121,A -85,B 0,C 180,E1 -9385.004,E2 -9385.004} C_VEL
LIN {X 0,Y 432.349,Z 233.126,A -85,B 0,C 180,E1 -9388.128,E2 -9388.128} C_VEL
LIN {X 0,Y 432.329,Z 233.125,A -85,B 0,C 180,E1 -9391.348,E2 -9391.348} C_VEL
LIN {X 0,Y 432.337,Z 233.129,A -85,B 0,C 180,E1 -9394.68,E2 -9394.68} C_VEL
LIN {X 0,Y 432.34,Z 233.124,A -85,B 0,C 180,E1 -9398.152,E2 -9398.152} C_VEL
LIN {X 0,Y 432.32,Z 233.128,A -85,B 0,C 180,E1 -9401.801,E2 -9401.801} C_VEL
LIN {X 0,Y 432.343,Z 233.127,A -85,B 0,C 180,E1 -9404.349,E2 -9404.349} C_VEL
LIN {X 0,Y 432.317,Z 233.128,A -85,B 0,C 180,E1 -9407.019,E2 -9407.019} C_VEL
LIN {X 0,Y 432.3,Z 233.137,A -85,B 0,C 180,E1 -9409.829,E2 -9409.829} C_VEL
LIN {X 0,Y 432.315,Z 233.131,A -85,B 0,C 180,E1 -9413.022,E2 -9413.022} C_VEL
LIN {X 0,Y 432.37,Z 233.125,A -85,B 0,C 180,E1 -9415.997,E2 -9415.997} C_VEL
LIN {X 0,Y 432.358,Z 233.125,A -85,B 0,C 180,E1 -9419.49,E2 -9419.49} C_VEL
LIN {X 0,Y 432.391,Z 233.123,A -85,B 0,C 180,E1 -9421.877,E2 -9421.877} C_VEL
LIN {X 0,Y 432.402,Z 233.234,A -85,B 0,C 180,E1 -9423.969,E2 -9423.969} C_VEL
LIN {X 0,Y 434.489,Z 243.953,A -85,B 0,C 180,E1 -9426.4,E2 -9426.4} C_VEL
LIN {X 0,Y 434.913,Z 247.589,A -85,B 0,C 180,E1 -9427.18,E2 -9427.18} C_VEL
LIN {X 0,Y 433.89,Z 264.479,A -85,B 0,C 180,E1 -9430.606,E2 -9430.606} C_VEL
LIN {X 0,Y 433.617,Z 269.678,A -85,B 0,C 180,E1 -9431.607,E2 -9431.607} C_VEL
LIN {X 0,Y 437.246,Z 291.665,A -85,B 0,C 180,E1 -9432.164,E2 -9432.164} C_VEL
LIN {X 0,Y 436.345,Z 376.918,A -85,B 0,C 180,E1 -9433.598,E2 -9433.598} C_VEL
LIN {X 0,Y 435.89,Z 390.312,A -85,B 0,C 180,E1 -9434.001,E2 -9434.001} C_VEL
LIN {X 0,Y 435.355,Z 403.668,A -85,B 0,C 180,E1 -9434.611,E2 -9434.611} C_VEL
LIN {X 0,Y 434.69,Z 415.664,A -85,B 0,C 180,E1 -9435.367,E2 -9435.367} C_VEL
LIN {X 0,Y 434.026,Z 427.209,A -85,B 0,C 180,E1 -9436.307,E2 -9436.307} C_VEL
LIN {X 0,Y 433.456,Z 437.493,A -85,B 0,C 180,E1 -9437.356,E2 -9437.356} C_VEL
LIN {X 0,Y 432.781,Z 446.777,A -85,B 0,C 180,E1 -9438.525,E2 -9438.525} C_VEL
LIN {X 0,Y 432.222,Z 455.788,A -85,B 0,C 180,E1 -9439.932,E2 -9439.932} C_VEL
LIN {X 0,Y 431.815,Z 463.043,A -85,B 0,C 180,E1 -9441.341,E2 -9441.341} C_VEL
LIN {X 0,Y 431.548,Z 467.941,A -85,B 0,C 180,E1 -9442.513,E2 -9442.513} C_VEL
LIN {X 0,Y 431.317,Z 472.915,A -85,B 0,C 180,E1 -9443.991,E2 -9443.991} C_VEL
LIN {X 0,Y 431.279,Z 476.337,A -85,B 0,C 180,E1 -9445.326,E2 -9445.326} C_VEL
LIN {X 0,Y 431.171,Z 478.216,A -85,B 0,C 180,E1 -9446.261,E2 -9446.261} C_VEL
LIN {X 0,Y 431.192,Z 479.63,A -85,B 0,C 180,E1 -9447.197,E2 -9447.197} C_VEL
LIN {X 0,Y 431.2,Z 480.636,A -85,B 0,C 180,E1 -9448.131,E2 -9448.131} C_VEL
LIN {X 0,Y 431.147,Z 481.48,A -85,B 0,C 180,E1 -9449.999,E2 -9449.999} C_VEL
LIN {X 0,Y 431.151,Z 481.278,A -85,B 0,C 180,E1 -9450.933,E2 -9450.933} C_VEL
LIN {X 0,Y 431.2,Z 480.678,A -85,B 0,C 180,E1 -9451.867,E2 -9451.867} C_VEL
LIN {X 0,Y 431.192,Z 479.69,A -85,B 0,C 180,E1 -9452.802,E2 -9452.802} C_VEL
LIN {X 0,Y 431.171,Z 478.304,A -85,B 0,C 180,E1 -9453.737,E2 -9453.737} C_VEL
LIN {X 0,Y 431.334,Z 475.382,A -85,B 0,C 180,E1 -9455.141,E2 -9455.141} C_VEL
LIN {X 0,Y 431.39,Z 471.425,A -85,B 0,C 180,E1 -9456.547,E2 -9456.547} C_VEL
LIN {X 0,Y 431.702,Z 465.343,A -85,B 0,C 180,E1 -9458.189,E2 -9458.189} C_VEL
LIN {X 0,Y 432.079,Z 458.688,A -85,B 0,C 180,E1 -9459.596,E2 -9459.596} C_VEL
LIN {X 0,Y 432.571,Z 450.429,A -85,B 0,C 180,E1 -9461.005,E2 -9461.005} C_VEL
LIN {X 0,Y 433.206,Z 441.973,A -85,B 0,C 180,E1 -9462.174,E2 -9462.174} C_VEL
LIN {X 0,Y 433.895,Z 432.145,A -85,B 0,C 180,E1 -9463.281,E2 -9463.281} C_VEL
LIN {X 0,Y 434.36,Z 422.62,A -85,B 0,C 180,E1 -9464.165,E2 -9464.165} C_VEL
LIN {X 0,Y 435.052,Z 411.646,A -85,B 0,C 180,E1 -9464.978,E2 -9464.978} C_VEL
LIN {X 0,Y 435.664,Z 399.507,A -85,B 0,C 180,E1 -9465.676,E2 -9465.676} C_VEL
LIN {X 0,Y 436.232,Z 386.911,A -85,B 0,C 180,E1 -9466.195,E2 -9466.195} C_VEL
LIN {X 0,Y 436.556,Z 373.758,A -85,B 0,C 180,E1 -9466.543,E2 -9466.543} C_VEL
LIN {X 0,Y 437.365,Z 290.847,A -85,B 0,C 180,E1 -9467.941,E2 -9467.941} C_VEL
LIN {X 0,Y 433.709,Z 269.59,A -85,B 0,C 180,E1 -9468.496,E2 -9468.496} C_VEL
LIN {X 0,Y 433.835,Z 265.964,A -85,B 0,C 180,E1 -9469.149,E2 -9469.149} C_VEL
LIN {X 0,Y 434.901,Z 247.609,A -85,B 0,C 180,E1 -9472.819,E2 -9472.819} C_VEL
LIN {X 0,Y 434.289,Z 242.709,A -85,B 0,C 180,E1 -9473.863,E2 -9473.863} C_VEL
LIN {X 0,Y 432.435,Z 233.341,A -85,B 0,C 180,E1 -9475.962,E2 -9475.962} C_VEL
LIN {X 0,Y 432.379,Z 233.127,A -85,B 0,C 180,E1 -9478.627,E2 -9478.627} C_VEL
LIN {X 0,Y 432.325,Z 233.133,A -85,B 0,C 180,E1 -9481.345,E2 -9481.345} C_VEL
LIN {X 0,Y 432.343,Z 233.13,A -85,B 0,C 180,E1 -9484.675,E2 -9484.675} C_VEL
LIN {X 0,Y 432.333,Z 233.135,A -85,B 0,C 180,E1 -9488.149,E2 -9488.149} C_VEL
LIN {X 0,Y 432.323,Z 233.131,A -85,B 0,C 180,E1 -9491.797,E2 -9491.797} C_VEL
LIN {X 0,Y 432.335,Z 233.135,A -85,B 0,C 180,E1 -9494.346,E2 -9494.346} C_VEL
LIN {X 0,Y 432.319,Z 233.131,A -85,B 0,C 180,E1 -9497.014,E2 -9497.014} C_VEL
LIN {X 0,Y 432.293,Z 233.134,A -85,B 0,C 180,E1 -9499.825,E2 -9499.825} C_VEL
LIN {X 0,Y 432.305,Z 233.134,A -85,B 0,C 180,E1 -9503.019,E2 -9503.019} C_VEL
LIN {X 0,Y 432.333,Z 233.128,A -85,B 0,C 180,E1 -9506,E2 -9506} C_VEL
LIN {X 0,Y 432.346,Z 233.126,A -85,B 0,C 180,E1 -9509.488,E2 -9509.488} C_VEL
LIN {X 0,Y 432.327,Z 233.127,A -85,B 0,C 180,E1 -9511.87,E2 -9511.87} C_VEL
LIN {X 0,Y 432.352,Z 233.125,A -85,B 0,C 180,E1 -9515.543,E2 -9515.543} C_VEL
LIN {X 0,Y 432.347,Z 233.133,A -85,B 0,C 180,E1 -9519.043,E2 -9519.043} C_VEL
LIN {X 0,Y 432.355,Z 233.119,A -85,B 0,C 180,E1 -9522.008,E2 -9522.008} C_VEL
LIN {X 0,Y 432.386,Z 233.127,A -85,B 0,C 180,E1 -9524.923,E2 -9524.923} C_VEL
LIN {X 0,Y 432.453,Z 233.113,A -85,B 0,C 180,E1 -9527.8,E2 -9527.8} C_VEL
LIN {X 0,Y 432.441,Z 233.114,A -85,B 0,C 180,E1 -9531.586,E2 -9531.586} C_VEL
LIN {X 0,Y 432.575,Z 233.098,A -85,B 0,C 180,E1 -9534.403,E2 -9534.403} C_VEL
LIN {X 0,Y 432.584,Z 233.098,A -85,B 0,C 180,E1 -9538.135,E2 -9538.135} C_VEL
LIN {X 0,Y 432.454,Z 233.11,A -85,B 0,C 180,E1 -9540.928,E2 -9540.928} C_VEL
LIN {X 0,Y 432.535,Z 233.102,A -85,B 0,C 180,E1 -9542.791,E2 -9542.791} C_VEL
LIN {X 0,Y 432.493,Z 233.107,A -85,B 0,C 180,E1 -9546.479,E2 -9546.479} C_VEL
LIN {X 0,Y 432.406,Z 233.12,A -85,B 0,C 180,E1 -9549.35,E2 -9549.35} C_VEL
LIN {X 0,Y 432.415,Z 233.116,A -85,B 0,C 180,E1 -9552.8,E2 -9552.8} C_VEL
LIN {X 0,Y 432.394,Z 233.12,A -85,B 0,C 180,E1 -9556.475,E2 -9556.475} C_VEL
LIN {X 0,Y 432.32,Z 233.134,A -85,B 0,C 180,E1 -9559.957,E2 -9559.957} C_VEL
LIN {X 0,Y 432.297,Z 233.132,A -85,B 0,C 180,E1 -9562.961,E2 -9562.961} C_VEL
LIN {X 0,Y 432.318,Z 233.129,A -85,B 0,C 180,E1 -9564.999,E2 -9564.999} C_VEL
LIN {X 0,Y 432.325,Z 233.13,A -85,B 0,C 180,E1 -9568.123,E2 -9568.123} C_VEL
LIN {X 0,Y 432.296,Z 233.133,A -85,B 0,C 180,E1 -9571.343,E2 -9571.343} C_VEL
LIN {X 0,Y 432.315,Z 233.132,A -85,B 0,C 180,E1 -9574.674,E2 -9574.674} C_VEL
LIN {X 0,Y 432.325,Z 233.132,A -85,B 0,C 180,E1 -9578.146,E2 -9578.146} C_VEL
LIN {X 0,Y 432.345,Z 233.132,A -85,B 0,C 180,E1 -9581.605,E2 -9581.605} C_VEL
LIN {X 0,Y 432.359,Z 233.216,A -85,B 0,C 180,E1 -9583.209,E2 -9583.209} C_VEL
LIN {X 0,Y 434.254,Z 242.794,A -85,B 0,C 180,E1 -9585.399,E2 -9585.399} C_VEL
LIN {X 0,Y 434.141,Z 250.273,A -85,B 0,C 180,E1 -9586.951,E2 -9586.951} C_VEL
LIN {X 0,Y 433.799,Z 258.231,A -85,B 0,C 180,E1 -9588.535,E2 -9588.535} C_VEL
LIN {X 0,Y 437.422,Z 277.754,A -85,B 0,C 180,E1 -9589.076,E2 -9589.076} C_VEL
LIN {X 0,Y 436.515,Z 365.628,A -85,B 0,C 180,E1 -9590.57,E2 -9590.57} C_VEL
LIN {X 0,Y 436.105,Z 379.355,A -85,B 0,C 180,E1 -9590.995,E2 -9590.995} C_VEL
LIN {X 0,Y 435.644,Z 392.411,A -85,B 0,C 180,E1 -9591.605,E2 -9591.605} C_VEL
LIN {X 0,Y 435.049,Z 403.775,A -85,B 0,C 180,E1 -9592.325,E2 -9592.325} C_VEL
LIN {X 0,Y 434.351,Z 414.908,A -85,B 0,C 180,E1 -9593.226,E2 -9593.226} C_VEL
LIN {X 0,Y 433.636,Z 425.574,A -85,B 0,C 180,E1 -9594.307,E2 -9594.307} C_VEL
LIN {X 0,Y 433.024,Z 435.272,A -85,B 0,C 180,E1 -9595.539,E2 -9595.539} C_VEL
LIN {X 0,Y 432.5,Z 443.018,A -85,B 0,C 180,E1 -9596.742,E2 -9596.742} C_VEL
LIN {X 0,Y 432.002,Z 450.536,A -85,B 0,C 180,E1 -9598.177,E2 -9598.177} C_VEL
LIN {X 0,Y 431.69,Z 456.835,A -85,B 0,C 180,E1 -9599.691,E2 -9599.691} C_VEL
LIN {X 0,Y 431.416,Z 461.743,A -85,B 0,C 180,E1 -9601.223,E2 -9601.223} C_VEL
LIN {X 0,Y 431.218,Z 465.55,A -85,B 0,C 180,E1 -9602.85,E2 -9602.85} C_VEL
LIN {X 0,Y 431.102,Z 467.308,A -85,B 0,C 180,E1 -9603.887,E2 -9603.887} C_VEL
LIN {X 0,Y 431.025,Z 468.533,A -85,B 0,C 180,E1 -9604.918,E2 -9604.918} C_VEL
LIN {X 0,Y 431.005,Z 469.259,A -85,B 0,C 180,E1 -9605.944,E2 -9605.944} C_VEL
LIN {X 0,Y 430.97,Z 469.538,A -85,B 0,C 180,E1 -9606.961,E2 -9606.961} C_VEL
LIN {X 0,Y 430.995,Z 469.121,A -85,B 0,C 180,E1 -9608.338,E2 -9608.338} C_VEL
LIN {X 0,Y 431.089,Z 467.523,A -85,B 0,C 180,E1 -9609.98,E2 -9609.98} C_VEL
LIN {X 0,Y 431.241,Z 464.956,A -85,B 0,C 180,E1 -9611.471,E2 -9611.471} C_VEL
LIN {X 0,Y 431.401,Z 461.308,A -85,B 0,C 180,E1 -9612.949,E2 -9612.949} C_VEL
LIN {X 0,Y 431.606,Z 456.991,A -85,B 0,C 180,E1 -9614.271,E2 -9614.271} C_VEL
LIN {X 0,Y 431.12,Z 454.397,A -85,B 0,C 180,E1 -9614.974,E2 -9614.974} C_VEL
LIN {X 0,Y 428.55,Z 449.77,A -85,B 0,C 180,E1 -9616.093,E2 -9616.093} C_VEL
LIN {X 0,Y 426,Z 444.502,A -85,B 0,C 180,E1 -9617.172,E2 -9617.172} C_VEL
LIN {X 0,Y 425.554,Z 440.9,A -85,B 0,C 180,E1 -9617.802,E2 -9617.802} C_VEL
LIN {X 0,Y 426.16,Z 432.329,A -85,B 0,C 180,E1 -9619.068,E2 -9619.068} C_VEL
LIN {X 0,Y 426.857,Z 422.192,A -85,B 0,C 180,E1 -9620.285,E2 -9620.285} C_VEL
LIN {X 0,Y 427.581,Z 411.354,A -85,B 0,C 180,E1 -9621.321,E2 -9621.321} C_VEL
LIN {X 0,Y 428.299,Z 399.389,A -85,B 0,C 180,E1 -9622.221,E2 -9622.221} C_VEL
LIN {X 0,Y 428.786,Z 386.911,A -85,B 0,C 180,E1 -9622.94,E2 -9622.94} C_VEL
LIN {X 0,Y 429.298,Z 374.257,A -85,B 0,C 180,E1 -9623.45,E2 -9623.45} C_VEL
LIN {X 0,Y 429.644,Z 361.465,A -85,B 0,C 180,E1 -9623.779,E2 -9623.779} C_VEL
LIN {X 0,Y 430.44,Z 278.442,A -85,B 0,C 180,E1 -9625.194,E2 -9625.194} C_VEL
LIN {X 0,Y 426.818,Z 258.732,A -85,B 0,C 180,E1 -9625.722,E2 -9625.722} C_VEL
LIN {X 0,Y 427.14,Z 251.873,A -85,B 0,C 180,E1 -9627.171,E2 -9627.171} C_VEL
LIN {X 0,Y 427.449,Z 245.505,A -85,B 0,C 180,E1 -9628.588,E2 -9628.588} C_VEL
LIN {X 0,Y 426.255,Z 237.507,A -85,B 0,C 180,E1 -9630.473,E2 -9630.473} C_VEL
LIN {X 0,Y 425.526,Z 234.033,A -85,B 0,C 180,E1 -9631.361,E2 -9631.361} C_VEL
LIN {X 0,Y 425.522,Z 233.98,A -85,B 0,C 180,E1 -9632.841,E2 -9632.841} C_VEL
LIN {X 0,Y 425.492,Z 233.98,A -85,B 0,C 180,E1 -9636.64,E2 -9636.64} C_VEL
LIN {X 0,Y 425.366,Z 233.997,A -85,B 0,C 180,E1 -9639.511,E2 -9639.511} C_VEL
LIN {X 0,Y 425.369,Z 233.989,A -85,B 0,C 180,E1 -9642.911,E2 -9642.911} C_VEL
LIN {X 0,Y 425.327,Z 233.999,A -85,B 0,C 180,E1 -9646.607,E2 -9646.607} C_VEL
LIN {X 0,Y 425.295,Z 234.007,A -85,B 0,C 180,E1 -9649.638,E2 -9649.638} C_VEL
LIN {X 0,Y 425.255,Z 234.012,A -85,B 0,C 180,E1 -9652.341,E2 -9652.341} C_VEL
LIN {X 0,Y 425.288,Z 234.005,A -85,B 0,C 180,E1 -9654.66,E2 -9654.66} C_VEL
LIN {X 0,Y 425.241,Z 234.013,A -85,B 0,C 180,E1 -9657.566,E2 -9657.566} C_VEL
LIN {X 0,Y 425.261,Z 234.01,A -85,B 0,C 180,E1 -9660.764,E2 -9660.764} C_VEL
LIN {X 0,Y 425.262,Z 234.008,A -85,B 0,C 180,E1 -9664.287,E2 -9664.287} C_VEL
LIN {X 0,Y 425.245,Z 234.01,A -85,B 0,C 180,E1 -9667.698,E2 -9667.698} C_VEL
LIN {X 0,Y 425.217,Z 234.017,A -85,B 0,C 180,E1 -9670.518,E2 -9670.518} C_VEL
LIN {X 0,Y 425.223,Z 234.007,A -85,B 0,C 180,E1 -9673.353,E2 -9673.353} C_VEL
LIN {X 0,Y 425.234,Z 234.012,A -85,B 0,C 180,E1 -9676.047,E2 -9676.047} C_VEL
LIN {X 0,Y 425.226,Z 234.017,A -85,B 0,C 180,E1 -9678.622,E2 -9678.622} C_VEL
LIN {X 0,Y 425.261,Z 233.998,A -85,B 0,C 180,E1 -9681.103,E2 -9681.103} C_VEL
LIN {X 0,Y 425.278,Z 234.006,A -85,B 0,C 180,E1 -9684.667,E2 -9684.667} C_VEL
LIN {X 0,Y 425.245,Z 234.007,A -85,B 0,C 180,E1 -9688.076,E2 -9688.076} C_VEL
LIN {X 0,Y 425.282,Z 233.992,A -85,B 0,C 180,E1 -9691.369,E2 -9691.369} C_VEL
LIN {X 0,Y 425.245,Z 234.006,A -85,B 0,C 180,E1 -9694.556,E2 -9694.556} C_VEL
LIN {X 0,Y 425.283,Z 234.008,A -85,B 0,C 180,E1 -9697.734,E2 -9697.734} C_VEL
LIN {X 0,Y 425.353,Z 233.986,A -85,B 0,C 180,E1 -9700.708,E2 -9700.708} C_VEL
LIN {X 0,Y 425.381,Z 233.98,A -85,B 0,C 180,E1 -9703.692,E2 -9703.692} C_VEL
LIN {X 0,Y 425.405,Z 233.994,A -85,B 0,C 180,E1 -9707.602,E2 -9707.602} C_VEL
LIN {X 0,Y 425.395,Z 233.989,A -85,B 0,C 180,E1 -9711.453,E2 -9711.453} C_VEL
LIN {X 0,Y 425.509,Z 233.962,A -85,B 0,C 180,E1 -9714.316,E2 -9714.316} C_VEL
LIN {X 0,Y 425.567,Z 233.973,A -85,B 0,C 180,E1 -9718.111,E2 -9718.111} C_VEL
LIN {X 0,Y 425.502,Z 233.976,A -85,B 0,C 180,E1 -9720.95,E2 -9720.95} C_VEL
LIN {X 0,Y 425.514,Z 233.969,A -85,B 0,C 180,E1 -9722.843,E2 -9722.843} C_VEL
LIN {X 0,Y 425.54,Z 233.955,A -85,B 0,C 180,E1 -9725.69,E2 -9725.69} C_VEL
LIN {X 0,Y 425.41,Z 233.993,A -85,B 0,C 180,E1 -9728.554,E2 -9728.554} C_VEL
LIN {X 0,Y 425.418,Z 233.993,A -85,B 0,C 180,E1 -9732.404,E2 -9732.404} C_VEL
LIN {X 0,Y 425.395,Z 233.98,A -85,B 0,C 180,E1 -9736.314,E2 -9736.314} C_VEL
LIN {X 0,Y 425.337,Z 233.999,A -85,B 0,C 180,E1 -9739.638,E2 -9739.638} C_VEL
LIN {X 0,Y 425.297,Z 234.003,A -85,B 0,C 180,E1 -9742.341,E2 -9742.341} C_VEL
LIN {X 0,Y 425.328,Z 233.99,A -85,B 0,C 180,E1 -9744.659,E2 -9744.659} C_VEL
LIN {X 0,Y 425.275,Z 234.009,A -85,B 0,C 180,E1 -9747.565,E2 -9747.565} C_VEL
LIN {X 0,Y 425.298,Z 234.002,A -85,B 0,C 180,E1 -9750.818,E2 -9750.818} C_VEL
LIN {X 0,Y 425.301,Z 234.004,A -85,B 0,C 180,E1 -9754.285,E2 -9754.285} C_VEL
LIN {X 0,Y 425.286,Z 234.005,A -85,B 0,C 180,E1 -9757.696,E2 -9757.696} C_VEL
LIN {X 0,Y 425.256,Z 234.009,A -85,B 0,C 180,E1 -9760.516,E2 -9760.516} C_VEL
LIN {X 0,Y 425.26,Z 234.008,A -85,B 0,C 180,E1 -9763.351,E2 -9763.351} C_VEL
LIN {X 0,Y 425.268,Z 234.008,A -85,B 0,C 180,E1 -9766.044,E2 -9766.044} C_VEL
LIN {X 0,Y 425.262,Z 234.009,A -85,B 0,C 180,E1 -9768.619,E2 -9768.619} C_VEL
LIN {X 0,Y 425.291,Z 234.007,A -85,B 0,C 180,E1 -9771.1,E2 -9771.1} C_VEL
LIN {X 0,Y 425.31,Z 234.005,A -85,B 0,C 180,E1 -9774.664,E2 -9774.664} C_VEL
LIN {X 0,Y 425.276,Z 234.015,A -85,B 0,C 180,E1 -9778.073,E2 -9778.073} C_VEL
LIN {X 0,Y 425.342,Z 234.001,A -85,B 0,C 180,E1 -9781.368,E2 -9781.368} C_VEL
LIN {X 0,Y 425.382,Z 234.194,A -85,B 0,C 180,E1 -9783.771,E2 -9783.771} C_VEL
LIN {X 0,Y 427.723,Z 246.229,A -85,B 0,C 180,E1 -9786.518,E2 -9786.518} C_VEL
LIN {X 0,Y 427.888,Z 249.997,A -85,B 0,C 180,E1 -9787.323,E2 -9787.323} C_VEL
LIN {X 0,Y 426.831,Z 266.754,A -85,B 0,C 180,E1 -9790.772,E2 -9790.772} C_VEL
LIN {X 0,Y 426.716,Z 269.68,A -85,B 0,C 180,E1 -9791.316,E2 -9791.316} C_VEL
LIN {X 0,Y 430.498,Z 292.782,A -85,B 0,C 180,E1 -9791.904,E2 -9791.904} C_VEL
LIN {X 0,Y 429.505,Z 377.618,A -85,B 0,C 180,E1 -9793.36,E2 -9793.36} C_VEL
LIN {X 0,Y 428.992,Z 391.492,A -85,B 0,C 180,E1 -9793.798,E2 -9793.798} C_VEL
LIN {X 0,Y 428.453,Z 404.451,A -85,B 0,C 180,E1 -9794.418,E2 -9794.418} C_VEL
LIN {X 0,Y 427.708,Z 417.023,A -85,B 0,C 180,E1 -9795.244,E2 -9795.244} C_VEL
LIN {X 0,Y 427.027,Z 428.077,A -85,B 0,C 180,E1 -9796.178,E2 -9796.178} C_VEL
LIN {X 0,Y 426.499,Z 437.311,A -85,B 0,C 180,E1 -9797.146,E2 -9797.146} C_VEL
LIN {X 0,Y 425.814,Z 446.616,A -85,B 0,C 180,E1 -9798.335,E2 -9798.335} C_VEL
LIN {X 0,Y 425.21,Z 455.637,A -85,B 0,C 180,E1 -9799.765,E2 -9799.765} C_VEL
LIN {X 0,Y 424.764,Z 462.903,A -85,B 0,C 180,E1 -9801.196,E2 -9801.196} C_VEL
LIN {X 0,Y 424.484,Z 467.81,A -85,B 0,C 180,E1 -9802.388,E2 -9802.388} C_VEL
LIN {X 0,Y 424.264,Z 472.174,A -85,B 0,C 180,E1 -9803.684,E2 -9803.684} C_VEL
LIN {X 0,Y 424.211,Z 476.221,A -85,B 0,C 180,E1 -9805.248,E2 -9805.248} C_VEL
LIN {X 0,Y 424.085,Z 478.103,A -85,B 0,C 180,E1 -9806.198,E2 -9806.198} C_VEL
LIN {X 0,Y 424.089,Z 479.522,A -85,B 0,C 180,E1 -9807.15,E2 -9807.15} C_VEL
LIN {X 0,Y 424.125,Z 480.531,A -85,B 0,C 180,E1 -9808.1,E2 -9808.1} C_VEL
LIN {X 0,Y 424.065,Z 481.382,A -85,B 0,C 180,E1 -9809.999,E2 -9809.999} C_VEL
LIN {X 0,Y 424.072,Z 481.183,A -85,B 0,C 180,E1 -9810.949,E2 -9810.949} C_VEL
LIN {X 0,Y 424.125,Z 480.586,A -85,B 0,C 180,E1 -9811.898,E2 -9811.898} C_VEL
LIN {X 0,Y 424.085,Z 478.216,A -85,B 0,C 180,E1 -9813.8,E2 -9813.8} C_VEL
LIN {X 0,Y 424.247,Z 475.298,A -85,B 0,C 180,E1 -9815.227,E2 -9815.227} C_VEL
LIN {X 0,Y 424.314,Z 471.344,A -85,B 0,C 180,E1 -9816.657,E2 -9816.657} C_VEL
LIN {X 0,Y 424.649,Z 465.27,A -85,B 0,C 180,E1 -9818.326,E2 -9818.326} C_VEL
LIN {X 0,Y 425.044,Z 458.619,A -85,B 0,C 180,E1 -9819.757,E2 -9819.757} C_VEL
LIN {X 0,Y 425.587,Z 450.365,A -85,B 0,C 180,E1 -9821.187,E2 -9821.187} C_VEL
LIN {X 0,Y 426.252,Z 441.923,A -85,B 0,C 180,E1 -9822.376,E2 -9822.376} C_VEL
LIN {X 0,Y 426.936,Z 432.453,A -85,B 0,C 180,E1 -9823.467,E2 -9823.467} C_VEL
LIN {X 0,Y 427.476,Z 422.614,A -85,B 0,C 180,E1 -9824.398,E2 -9824.398} C_VEL
LIN {X 0,Y 428.212,Z 411.671,A -85,B 0,C 180,E1 -9825.223,E2 -9825.223} C_VEL
LIN {X 0,Y 428.849,Z 399.578,A -85,B 0,C 180,E1 -9825.931,E2 -9825.931} C_VEL
LIN {X 0,Y 429.427,Z 387.099,A -85,B 0,C 180,E1 -9826.458,E2 -9826.458} C_VEL
LIN {X 0,Y 429.781,Z 374.134,A -85,B 0,C 180,E1 -9826.811,E2 -9826.811} C_VEL
LIN {X 0,Y 430.68,Z 292.007,A -85,B 0,C 180,E1 -9828.218,E2 -9828.218} C_VEL
LIN {X 0,Y 426.786,Z 269.288,A -85,B 0,C 180,E1 -9828.837,E2 -9828.837} C_VEL
LIN {X 0,Y 427.725,Z 252.451,A -85,B 0,C 180,E1 -9832.204,E2 -9832.204} C_VEL
LIN {X 0,Y 427.916,Z 247.558,A -85,B 0,C 180,E1 -9833.213,E2 -9833.213} C_VEL
LIN {X 0,Y 425.643,Z 235.339,A -85,B 0,C 180,E1 -9835.947,E2 -9835.947} C_VEL
LIN {X 0,Y 425.354,Z 234.031,A -85,B 0,C 180,E1 -9836.328,E2 -9836.328} C_VEL
LIN {X 0,Y 425.296,Z 234.009,A -85,B 0,C 180,E1 -9839.718,E2 -9839.718} C_VEL
LIN {X 0,Y 425.287,Z 234.009,A -85,B 0,C 180,E1 -9843.046,E2 -9843.046} C_VEL
LIN {X 0,Y 425.285,Z 234.009,A -85,B 0,C 180,E1 -9845.926,E2 -9845.926} C_VEL
LIN {X 0,Y 425.265,Z 234.008,A -85,B 0,C 180,E1 -9849.035,E2 -9849.035} C_VEL
LIN {X 0,Y 425.272,Z 234.009,A -85,B 0,C 180,E1 -9852.652,E2 -9852.652} C_VEL
LIN {X 0,Y 425.263,Z 234.011,A -85,B 0,C 180,E1 -9856.042,E2 -9856.042} C_VEL
LIN {X 0,Y 425.259,Z 234.013,A -85,B 0,C 180,E1 -9858.617,E2 -9858.617} C_VEL
LIN {X 0,Y 425.282,Z 234.004,A -85,B 0,C 180,E1 -9861.097,E2 -9861.097} C_VEL
LIN {X 0,Y 425.296,Z 234.006,A -85,B 0,C 180,E1 -9864.661,E2 -9864.661} C_VEL
LIN {X 0,Y 425.263,Z 234.009,A -85,B 0,C 180,E1 -9868.07,E2 -9868.07} C_VEL
LIN {X 0,Y 425.304,Z 234.003,A -85,B 0,C 180,E1 -9871.363,E2 -9871.363} C_VEL
LIN {X 0,Y 425.258,Z 234.012,A -85,B 0,C 180,E1 -9874.55,E2 -9874.55} C_VEL
LIN {X 0,Y 425.29,Z 234.003,A -85,B 0,C 180,E1 -9877.727,E2 -9877.727} C_VEL
LIN {X 0,Y 425.358,Z 234,A -85,B 0,C 180,E1 -9880.701,E2 -9880.701} C_VEL
LIN {X 0,Y 425.384,Z 233.995,A -85,B 0,C 180,E1 -9883.685,E2 -9883.685} C_VEL
LIN {X 0,Y 425.407,Z 233.993,A -85,B 0,C 180,E1 -9887.595,E2 -9887.595} C_VEL
LIN {X 0,Y 425.389,Z 233.992,A -85,B 0,C 180,E1 -9891.446,E2 -9891.446} C_VEL
LIN {X 0,Y 425.531,Z 233.975,A -85,B 0,C 180,E1 -9894.31,E2 -9894.31} C_VEL
LIN {X 0,Y 425.553,Z 233.974,A -85,B 0,C 180,E1 -9898.104,E2 -9898.104} C_VEL
LIN {X 0,Y 425.424,Z 233.986,A -85,B 0,C 180,E1 -9900.943,E2 -9900.943} C_VEL
LIN {X 0,Y 425.492,Z 233.98,A -85,B 0,C 180,E1 -9902.837,E2 -9902.837} C_VEL
LIN {X 0,Y 425.454,Z 233.983,A -85,B 0,C 180,E1 -9906.48,E2 -9906.48} C_VEL
LIN {X 0,Y 425.367,Z 233.998,A -85,B 0,C 180,E1 -9909.507,E2 -9909.507} C_VEL
LIN {X 0,Y 425.378,Z 233.993,A -85,B 0,C 180,E1 -9912.9,E2 -9912.9} C_VEL
LIN {X 0,Y 425.344,Z 233.997,A -85,B 0,C 180,E1 -9916.601,E2 -9916.601} C_VEL
LIN {X 0,Y 425.31,Z 234.006,A -85,B 0,C 180,E1 -9919.632,E2 -9919.632} C_VEL
LIN {X 0,Y 425.268,Z 234.011,A -85,B 0,C 180,E1 -9922.336,E2 -9922.336} C_VEL
LIN {X 0,Y 425.299,Z 234.006,A -85,B 0,C 180,E1 -9924.654,E2 -9924.654} C_VEL
LIN {X 0,Y 425.25,Z 234.011,A -85,B 0,C 180,E1 -9927.56,E2 -9927.56} C_VEL
LIN {X 0,Y 425.267,Z 234.012,A -85,B 0,C 180,E1 -9930.758,E2 -9930.758} C_VEL
LIN {X 0,Y 425.287,Z 234.011,A -85,B 0,C 180,E1 -9934.285,E2 -9934.285} C_VEL
LIN {X 0,Y 425.261,Z 234.01,A -85,B 0,C 180,E1 -9937.691,E2 -9937.691} C_VEL
LIN {X 0,Y 425.274,Z 234.013,A -85,B 0,C 180,E1 -9940.521,E2 -9940.521} C_VEL
LIN {X 0,Y 425.314,Z 234.073,A -85,B 0,C 180,E1 -9942.945,E2 -9942.945} C_VEL
LIN {X 0,Y 427.348,Z 244.297,A -85,B 0,C 180,E1 -9945.324,E2 -9945.324} C_VEL
LIN {X 0,Y 427.171,Z 251.98,A -85,B 0,C 180,E1 -9946.941,E2 -9946.941} C_VEL
LIN {X 0,Y 426.893,Z 258.303,A -85,B 0,C 180,E1 -9948.21,E2 -9948.21} C_VEL
LIN {X 0,Y 430.638,Z 278.158,A -85,B 0,C 180,E1 -9948.777,E2 -9948.777} C_VEL
LIN {X 0,Y 430.646,Z 293.803,A -85,B 0,C 180,E1 -9949.053,E2 -9949.053} C_VEL
LIN {X 0,Y 429.698,Z 366.562,A -85,B 0,C 180,E1 -9950.314,E2 -9950.314} C_VEL
LIN {X 0,Y 429.288,Z 380.346,A -85,B 0,C 180,E1 -9950.759,E2 -9950.759} C_VEL
LIN {X 0,Y 428.82,Z 392.299,A -85,B 0,C 180,E1 -9951.331,E2 -9951.331} C_VEL
LIN {X 0,Y 428.253,Z 403.51,A -85,B 0,C 180,E1 -9952.049,E2 -9952.049} C_VEL
LIN {X 0,Y 427.471,Z 414.869,A -85,B 0,C 180,E1 -9952.978,E2 -9952.978} C_VEL
LIN {X 0,Y 426.702,Z 425.75,A -85,B 0,C 180,E1 -9954.097,E2 -9954.097} C_VEL
LIN {X 0,Y 426.147,Z 434.535,A -85,B 0,C 180,E1 -9955.22,E2 -9955.22} C_VEL
LIN {X 0,Y 425.579,Z 442.259,A -85,B 0,C 180,E1 -9956.413,E2 -9956.413} C_VEL
LIN {X 0,Y 425.071,Z 449.369,A -85,B 0,C 180,E1 -9957.752,E2 -9957.752} C_VEL
LIN {X 0,Y 424.661,Z 456.223,A -85,B 0,C 180,E1 -9959.372,E2 -9959.372} C_VEL
LIN {X 0,Y 424.373,Z 460.805,A -85,B 0,C 180,E1 -9960.756,E2 -9960.756} C_VEL
LIN {X 0,Y 424.18,Z 464.842,A -85,B 0,C 180,E1 -9962.361,E2 -9962.361} C_VEL
LIN {X 0,Y 424.028,Z 466.909,A -85,B 0,C 180,E1 -9963.499,E2 -9963.499} C_VEL
LIN {X 0,Y 423.945,Z 468.209,A -85,B 0,C 180,E1 -9964.469,E2 -9964.469} C_VEL
LIN {X 0,Y 423.898,Z 469.275,A -85,B 0,C 180,E1 -9965.753,E2 -9965.753} C_VEL
LIN {X 0,Y 423.874,Z 469.546,A -85,B 0,C 180,E1 -9967.584,E2 -9967.584} C_VEL
LIN {X 0,Y 423.902,Z 469.064,A -85,B 0,C 180,E1 -9968.609,E2 -9968.609} C_VEL
LIN {X 0,Y 423.977,Z 468.088,A -85,B 0,C 180,E1 -9969.63,E2 -9969.63} C_VEL
LIN {X 0,Y 424.094,Z 466.399,A -85,B 0,C 180,E1 -9970.822,E2 -9970.822} C_VEL
LIN {X 0,Y 424.216,Z 463.683,A -85,B 0,C 180,E1 -9972.153,E2 -9972.153} C_VEL
LIN {X 0,Y 424.44,Z 459.1,A -85,B 0,C 180,E1 -9973.8,E2 -9973.8} C_VEL
LIN {X 0,Y 424.806,Z 453.191,A -85,B 0,C 180,E1 -9975.388,E2 -9975.388} C_VEL
LIN {X 0,Y 425.277,Z 445.657,A -85,B 0,C 180,E1 -9976.974,E2 -9976.974} C_VEL
LIN {X 0,Y 425.554,Z 440.9,A -85,B 0,C 180,E1 -9977.802,E2 -9977.802} C_VEL
LIN {X 0,Y 425.146,Z 437.134,A -85,B 0,C 180,E1 -9978.412,E2 -9978.412} C_VEL
LIN {X 0,Y 421.722,Z 428.061,A -85,B 0,C 180,E1 -9979.759,E2 -9979.759} C_VEL
LIN {X 0,Y 420.226,Z 422.371,A -85,B 0,C 180,E1 -9980.476,E2 -9980.476} C_VEL
LIN {X 0,Y 420.123,Z 419.264,A -85,B 0,C 180,E1 -9980.811,E2 -9980.811} C_VEL
LIN {X 0,Y 420.894,Z 407.966,A -85,B 0,C 180,E1 -9981.841,E2 -9981.841} C_VEL
LIN {X 0,Y 421.585,Z 395.804,A -85,B 0,C 180,E1 -9982.698,E2 -9982.698} C_VEL
LIN {X 0,Y 422.127,Z 383.145,A -85,B 0,C 180,E1 -9983.368,E2 -9983.368} C_VEL
LIN {X 0,Y 422.604,Z 370.739,A -85,B 0,C 180,E1 -9983.825,E2 -9983.825} C_VEL
LIN {X 0,Y 422.891,Z 355.175,A -85,B 0,C 180,E1 -9984.159,E2 -9984.159} C_VEL
LIN {X 0,Y 423.716,Z 279.619,A -85,B 0,C 180,E1 -9985.46,E2 -9985.46} C_VEL
LIN {X 0,Y 419.913,Z 258.905,A -85,B 0,C 180,E1 -9986.027,E2 -9986.027} C_VEL
LIN {X 0,Y 420.007,Z 255.795,A -85,B 0,C 180,E1 -9986.643,E2 -9986.643} C_VEL
LIN {X 0,Y 420.531,Z 247.25,A -85,B 0,C 180,E1 -9988.564,E2 -9988.564} C_VEL
LIN {X 0,Y 419.387,Z 239.234,A -85,B 0,C 180,E1 -9990.481,E2 -9990.481} C_VEL
LIN {X 0,Y 418.498,Z 234.908,A -85,B 0,C 180,E1 -9991.595,E2 -9991.595} C_VEL
